(* Logix 5000 project; controller CarbonScout_MK6 vendor 1 type 14 code 154 rev 32.11; software revision 32.00; part 16 of 17 *)
(* tags used below, declared in another part *)
   ONS : BOOL[32];
   a_Software_Version : STRING;   // This must be updated and have a corrosponding change log and compadibility doc
   CS_DINTParams : DINT[100];
   CS_Seq : GEK_Sequence;
   CS_XRF : XRF;
   CS_XRF_Elements : LinearModelXRF;   // Linear model 0 is inital factory model and 1 is trimming model
   CS_XRF_Elements_Saved : LinearModelXRF;
   CS_XRF_RawModel : REAL[4];
   N50 : DINT[20];   // Out To Client (Ready only)
   NetworkHealthy : DINT;
   Oneshot3 : DINT;
   PLC_Powered : BOOL;
   Powered_Up : TIMER;
   Reg_Model : REAL[4];   // Calculated model output and site model
   Simulation : DINT;
   TimeAndDate : DINT[7];
   TimeAndDateW : DINT[7];
   Uptime : DINT;   // sec
   Valve_XV_01 : P_ValveSO;   // Sample Valve Tank 1
   Valve_XV_02 : P_ValveSO;   // Sample Valve Tank 2
   Valve_XV_03 : P_ValveSO;   // Sample Valve Tank 3
   Valve_XV_04 : P_ValveSO;   // Sample Valve Tank 4
   Valve_XV_05 : P_ValveSO;   // Sample Valve Tank 5
   Valve_XV_06 : P_ValveSO;   // Sample Valve Tank 6
   Valve_XV_07 : P_ValveSO;   // Sample Valve Tank 7
   Valve_XV_08 : P_ValveSO;   // Sample Valve Tank 8
   Valve_XV_09 : P_ValveSO;   // Sample Valve Tank 9
   Valve_XV_10 : P_ValveSO;   // Sample Valve Tank 10
   Valve_XV_11 : P_ValveSO;   // Purge Valve
   Valve_XV_12 : P_ValveSO;   // Slurry inlet vavle
   Valve_XV_13 : P_ValveSO;   // Sample line vavle
   XRF_RAWDINT : DINT[100];
(* SeqProgram, continued *)

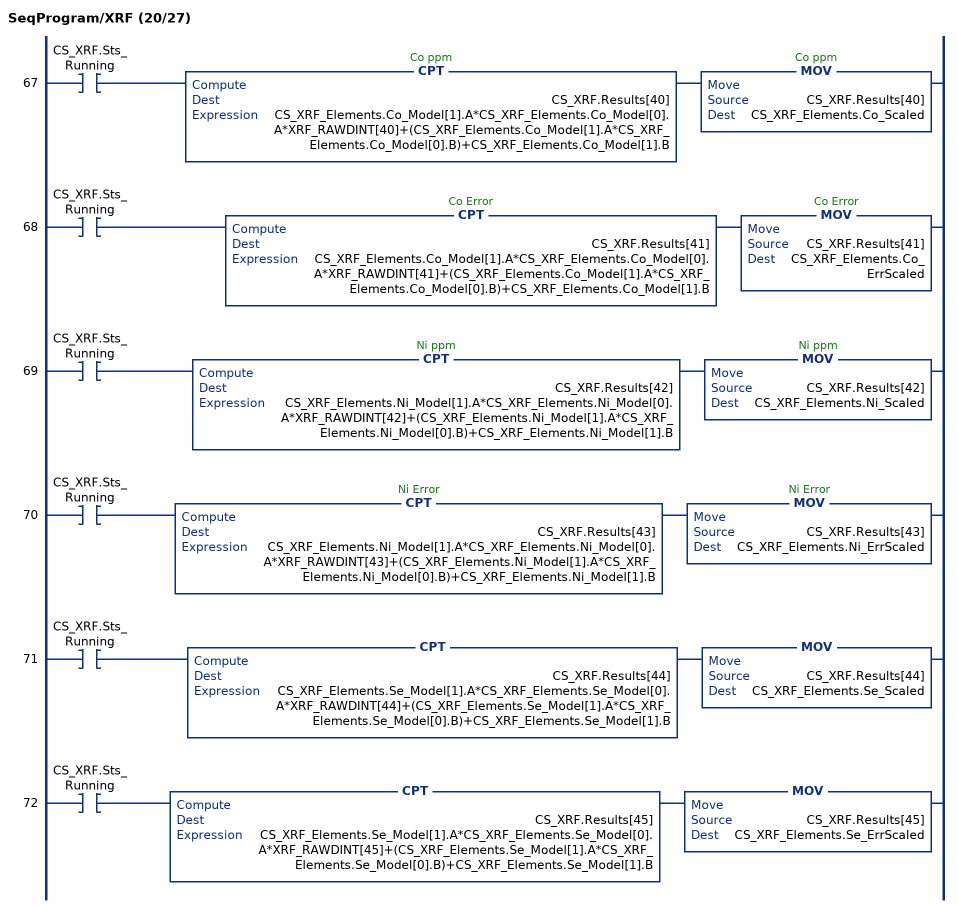
   67: XIC(CS_XRF.Sts_Running)CPT(CS_XRF.Results[40],CS_XRF_Elements.Co_Model[1].A*CS_XRF_Elements.Co_Model[0].A*XRF_RAWDINT[40]+(CS_XRF_Elements.Co_Model[1].A*CS_XRF_Elements.Co_Model[0].B)+CS_XRF_Elements.Co_Model[1].B)MOV(CS_XRF.Results[40],CS_XRF_Elements.Co_Scaled);
   68: XIC(CS_XRF.Sts_Running)CPT(CS_XRF.Results[41],CS_XRF_Elements.Co_Model[1].A*CS_XRF_Elements.Co_Model[0].A*XRF_RAWDINT[41]+(CS_XRF_Elements.Co_Model[1].A*CS_XRF_Elements.Co_Model[0].B)+CS_XRF_Elements.Co_Model[1].B)MOV(CS_XRF.Results[41],CS_XRF_Elements.Co_ErrScaled);
   69: XIC(CS_XRF.Sts_Running)CPT(CS_XRF.Results[42],CS_XRF_Elements.Ni_Model[1].A*CS_XRF_Elements.Ni_Model[0].A*XRF_RAWDINT[42]+(CS_XRF_Elements.Ni_Model[1].A*CS_XRF_Elements.Ni_Model[0].B)+CS_XRF_Elements.Ni_Model[1].B)MOV(CS_XRF.Results[42],CS_XRF_Elements.Ni_Scaled);
   70: XIC(CS_XRF.Sts_Running)CPT(CS_XRF.Results[43],CS_XRF_Elements.Ni_Model[1].A*CS_XRF_Elements.Ni_Model[0].A*XRF_RAWDINT[43]+(CS_XRF_Elements.Ni_Model[1].A*CS_XRF_Elements.Ni_Model[0].B)+CS_XRF_Elements.Ni_Model[1].B)MOV(CS_XRF.Results[43],CS_XRF_Elements.Ni_ErrScaled);
   71: XIC(CS_XRF.Sts_Running)CPT(CS_XRF.Results[44],CS_XRF_Elements.Se_Model[1].A*CS_XRF_Elements.Se_Model[0].A*XRF_RAWDINT[44]+(CS_XRF_Elements.Se_Model[1].A*CS_XRF_Elements.Se_Model[0].B)+CS_XRF_Elements.Se_Model[1].B)MOV(CS_XRF.Results[44],CS_XRF_Elements.Se_Scaled);
   72: XIC(CS_XRF.Sts_Running)CPT(CS_XRF.Results[45],CS_XRF_Elements.Se_Model[1].A*CS_XRF_Elements.Se_Model[0].A*XRF_RAWDINT[45]+(CS_XRF_Elements.Se_Model[1].A*CS_XRF_Elements.Se_Model[0].B)+CS_XRF_Elements.Se_Model[1].B)MOV(CS_XRF.Results[45],CS_XRF_Elements.Se_ErrScaled);
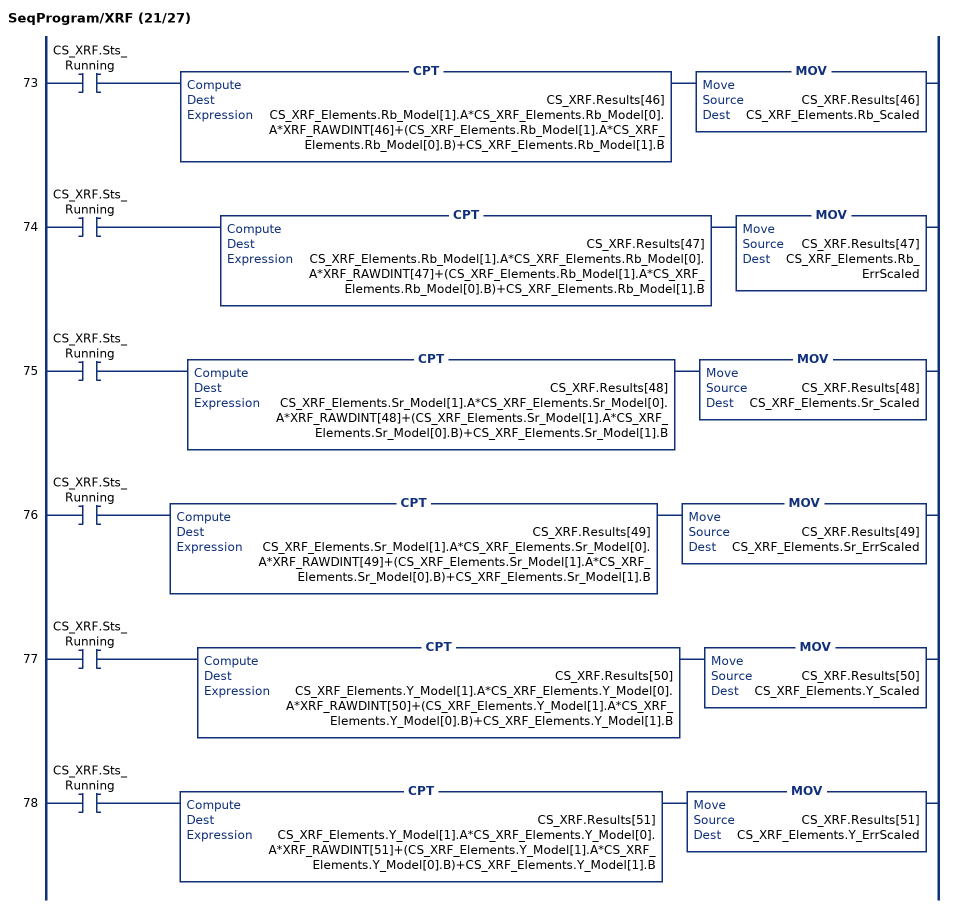
   73: XIC(CS_XRF.Sts_Running)CPT(CS_XRF.Results[46],CS_XRF_Elements.Rb_Model[1].A*CS_XRF_Elements.Rb_Model[0].A*XRF_RAWDINT[46]+(CS_XRF_Elements.Rb_Model[1].A*CS_XRF_Elements.Rb_Model[0].B)+CS_XRF_Elements.Rb_Model[1].B)MOV(CS_XRF.Results[46],CS_XRF_Elements.Rb_Scaled);
   74: XIC(CS_XRF.Sts_Running)CPT(CS_XRF.Results[47],CS_XRF_Elements.Rb_Model[1].A*CS_XRF_Elements.Rb_Model[0].A*XRF_RAWDINT[47]+(CS_XRF_Elements.Rb_Model[1].A*CS_XRF_Elements.Rb_Model[0].B)+CS_XRF_Elements.Rb_Model[1].B)MOV(CS_XRF.Results[47],CS_XRF_Elements.Rb_ErrScaled);
   75: XIC(CS_XRF.Sts_Running)CPT(CS_XRF.Results[48],CS_XRF_Elements.Sr_Model[1].A*CS_XRF_Elements.Sr_Model[0].A*XRF_RAWDINT[48]+(CS_XRF_Elements.Sr_Model[1].A*CS_XRF_Elements.Sr_Model[0].B)+CS_XRF_Elements.Sr_Model[1].B)MOV(CS_XRF.Results[48],CS_XRF_Elements.Sr_Scaled);
   76: XIC(CS_XRF.Sts_Running)CPT(CS_XRF.Results[49],CS_XRF_Elements.Sr_Model[1].A*CS_XRF_Elements.Sr_Model[0].A*XRF_RAWDINT[49]+(CS_XRF_Elements.Sr_Model[1].A*CS_XRF_Elements.Sr_Model[0].B)+CS_XRF_Elements.Sr_Model[1].B)MOV(CS_XRF.Results[49],CS_XRF_Elements.Sr_ErrScaled);
   77: XIC(CS_XRF.Sts_Running)CPT(CS_XRF.Results[50],CS_XRF_Elements.Y_Model[1].A*CS_XRF_Elements.Y_Model[0].A*XRF_RAWDINT[50]+(CS_XRF_Elements.Y_Model[1].A*CS_XRF_Elements.Y_Model[0].B)+CS_XRF_Elements.Y_Model[1].B)MOV(CS_XRF.Results[50],CS_XRF_Elements.Y_Scaled);
   78: XIC(CS_XRF.Sts_Running)CPT(CS_XRF.Results[51],CS_XRF_Elements.Y_Model[1].A*CS_XRF_Elements.Y_Model[0].A*XRF_RAWDINT[51]+(CS_XRF_Elements.Y_Model[1].A*CS_XRF_Elements.Y_Model[0].B)+CS_XRF_Elements.Y_Model[1].B)MOV(CS_XRF.Results[51],CS_XRF_Elements.Y_ErrScaled);
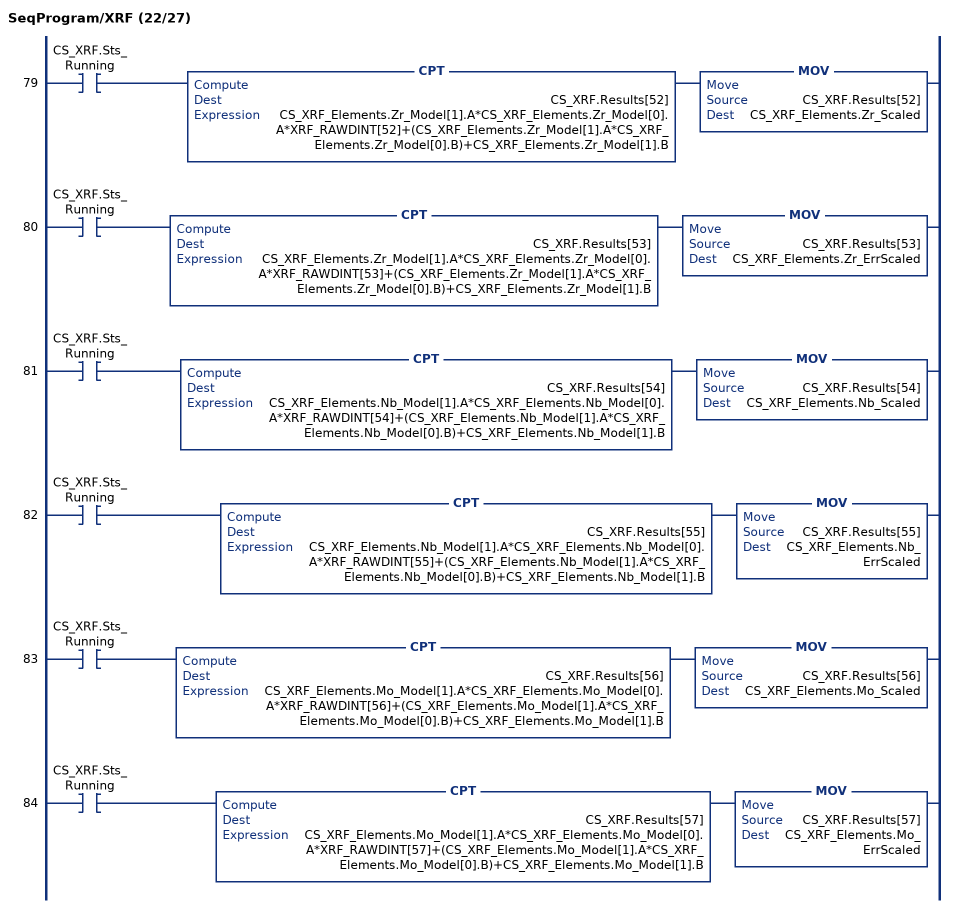
   79: XIC(CS_XRF.Sts_Running)CPT(CS_XRF.Results[52],CS_XRF_Elements.Zr_Model[1].A*CS_XRF_Elements.Zr_Model[0].A*XRF_RAWDINT[52]+(CS_XRF_Elements.Zr_Model[1].A*CS_XRF_Elements.Zr_Model[0].B)+CS_XRF_Elements.Zr_Model[1].B)MOV(CS_XRF.Results[52],CS_XRF_Elements.Zr_Scaled);
   80: XIC(CS_XRF.Sts_Running)CPT(CS_XRF.Results[53],CS_XRF_Elements.Zr_Model[1].A*CS_XRF_Elements.Zr_Model[0].A*XRF_RAWDINT[53]+(CS_XRF_Elements.Zr_Model[1].A*CS_XRF_Elements.Zr_Model[0].B)+CS_XRF_Elements.Zr_Model[1].B)MOV(CS_XRF.Results[53],CS_XRF_Elements.Zr_ErrScaled);
   81: XIC(CS_XRF.Sts_Running)CPT(CS_XRF.Results[54],CS_XRF_Elements.Nb_Model[1].A*CS_XRF_Elements.Nb_Model[0].A*XRF_RAWDINT[54]+(CS_XRF_Elements.Nb_Model[1].A*CS_XRF_Elements.Nb_Model[0].B)+CS_XRF_Elements.Nb_Model[1].B)MOV(CS_XRF.Results[54],CS_XRF_Elements.Nb_Scaled);
   82: XIC(CS_XRF.Sts_Running)CPT(CS_XRF.Results[55],CS_XRF_Elements.Nb_Model[1].A*CS_XRF_Elements.Nb_Model[0].A*XRF_RAWDINT[55]+(CS_XRF_Elements.Nb_Model[1].A*CS_XRF_Elements.Nb_Model[0].B)+CS_XRF_Elements.Nb_Model[1].B)MOV(CS_XRF.Results[55],CS_XRF_Elements.Nb_ErrScaled);
   83: XIC(CS_XRF.Sts_Running)CPT(CS_XRF.Results[56],CS_XRF_Elements.Mo_Model[1].A*CS_XRF_Elements.Mo_Model[0].A*XRF_RAWDINT[56]+(CS_XRF_Elements.Mo_Model[1].A*CS_XRF_Elements.Mo_Model[0].B)+CS_XRF_Elements.Mo_Model[1].B)MOV(CS_XRF.Results[56],CS_XRF_Elements.Mo_Scaled);
   84: XIC(CS_XRF.Sts_Running)CPT(CS_XRF.Results[57],CS_XRF_Elements.Mo_Model[1].A*CS_XRF_Elements.Mo_Model[0].A*XRF_RAWDINT[57]+(CS_XRF_Elements.Mo_Model[1].A*CS_XRF_Elements.Mo_Model[0].B)+CS_XRF_Elements.Mo_Model[1].B)MOV(CS_XRF.Results[57],CS_XRF_Elements.Mo_ErrScaled);
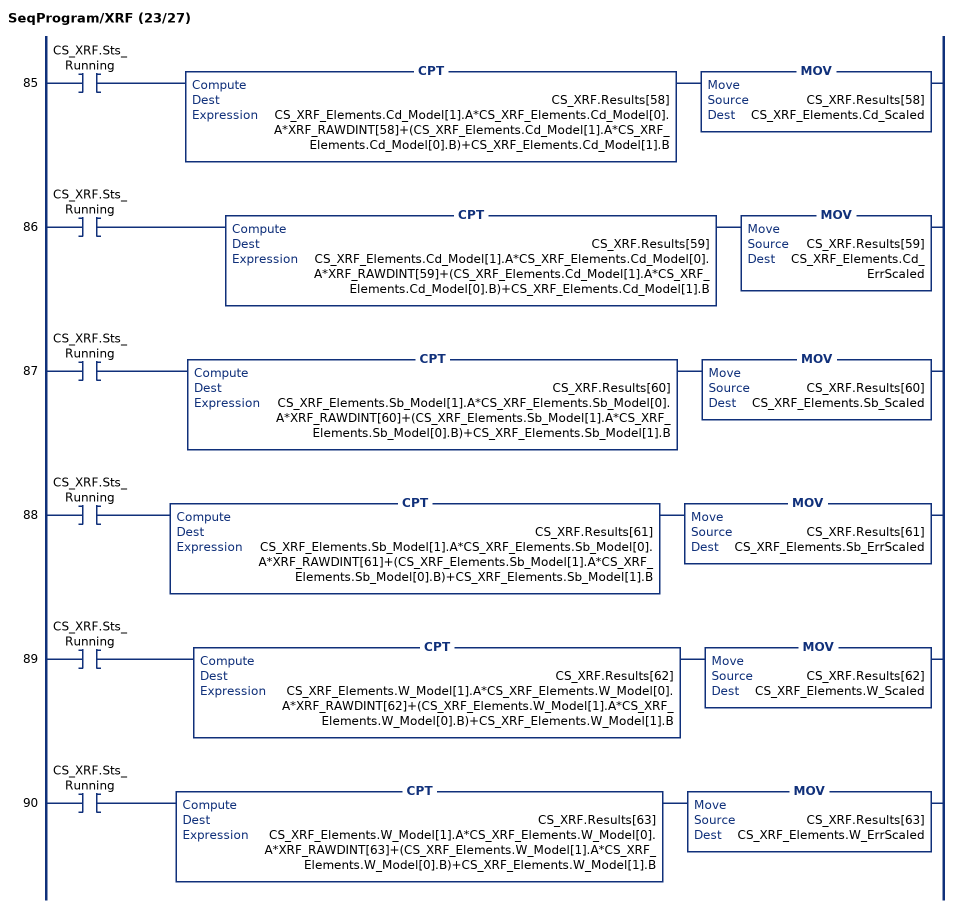
   85: XIC(CS_XRF.Sts_Running)CPT(CS_XRF.Results[58],CS_XRF_Elements.Cd_Model[1].A*CS_XRF_Elements.Cd_Model[0].A*XRF_RAWDINT[58]+(CS_XRF_Elements.Cd_Model[1].A*CS_XRF_Elements.Cd_Model[0].B)+CS_XRF_Elements.Cd_Model[1].B)MOV(CS_XRF.Results[58],CS_XRF_Elements.Cd_Scaled);
   86: XIC(CS_XRF.Sts_Running)CPT(CS_XRF.Results[59],CS_XRF_Elements.Cd_Model[1].A*CS_XRF_Elements.Cd_Model[0].A*XRF_RAWDINT[59]+(CS_XRF_Elements.Cd_Model[1].A*CS_XRF_Elements.Cd_Model[0].B)+CS_XRF_Elements.Cd_Model[1].B)MOV(CS_XRF.Results[59],CS_XRF_Elements.Cd_ErrScaled);
   87: XIC(CS_XRF.Sts_Running)CPT(CS_XRF.Results[60],CS_XRF_Elements.Sb_Model[1].A*CS_XRF_Elements.Sb_Model[0].A*XRF_RAWDINT[60]+(CS_XRF_Elements.Sb_Model[1].A*CS_XRF_Elements.Sb_Model[0].B)+CS_XRF_Elements.Sb_Model[1].B)MOV(CS_XRF.Results[60],CS_XRF_Elements.Sb_Scaled);
   88: XIC(CS_XRF.Sts_Running)CPT(CS_XRF.Results[61],CS_XRF_Elements.Sb_Model[1].A*CS_XRF_Elements.Sb_Model[0].A*XRF_RAWDINT[61]+(CS_XRF_Elements.Sb_Model[1].A*CS_XRF_Elements.Sb_Model[0].B)+CS_XRF_Elements.Sb_Model[1].B)MOV(CS_XRF.Results[61],CS_XRF_Elements.Sb_ErrScaled);
   89: XIC(CS_XRF.Sts_Running)CPT(CS_XRF.Results[62],CS_XRF_Elements.W_Model[1].A*CS_XRF_Elements.W_Model[0].A*XRF_RAWDINT[62]+(CS_XRF_Elements.W_Model[1].A*CS_XRF_Elements.W_Model[0].B)+CS_XRF_Elements.W_Model[1].B)MOV(CS_XRF.Results[62],CS_XRF_Elements.W_Scaled);
   90: XIC(CS_XRF.Sts_Running)CPT(CS_XRF.Results[63],CS_XRF_Elements.W_Model[1].A*CS_XRF_Elements.W_Model[0].A*XRF_RAWDINT[63]+(CS_XRF_Elements.W_Model[1].A*CS_XRF_Elements.W_Model[0].B)+CS_XRF_Elements.W_Model[1].B)MOV(CS_XRF.Results[63],CS_XRF_Elements.W_ErrScaled);
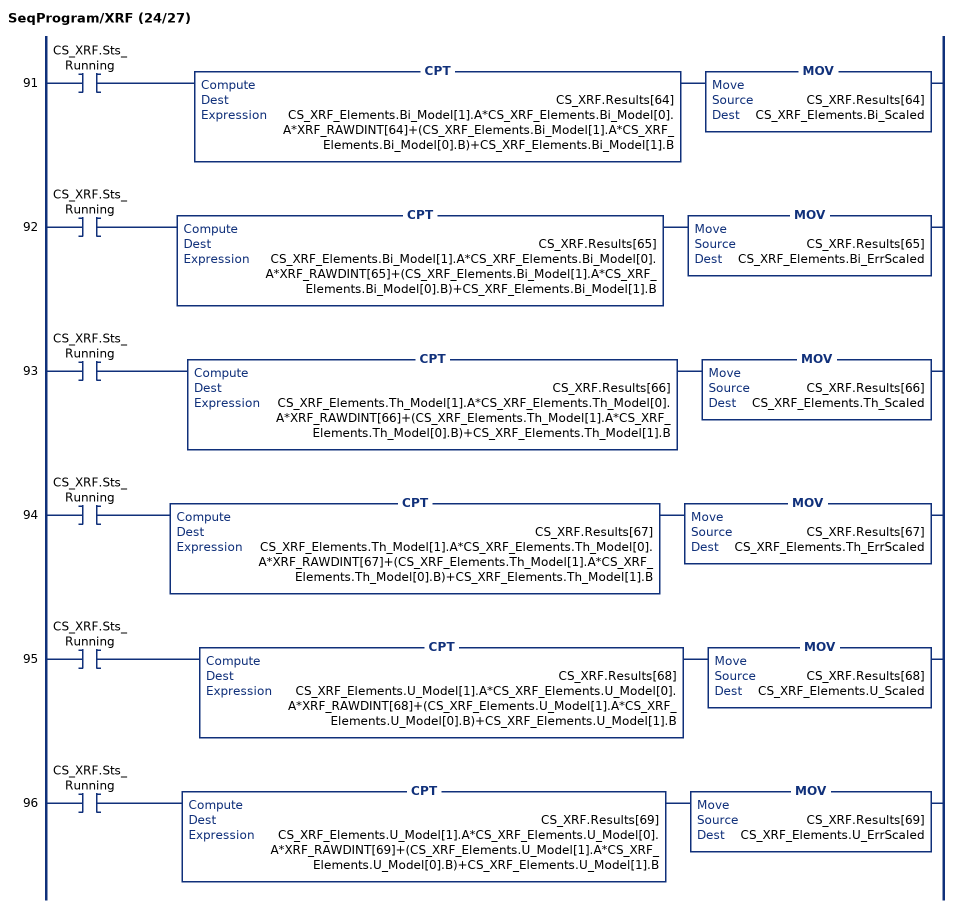
   91: XIC(CS_XRF.Sts_Running)CPT(CS_XRF.Results[64],CS_XRF_Elements.Bi_Model[1].A*CS_XRF_Elements.Bi_Model[0].A*XRF_RAWDINT[64]+(CS_XRF_Elements.Bi_Model[1].A*CS_XRF_Elements.Bi_Model[0].B)+CS_XRF_Elements.Bi_Model[1].B)MOV(CS_XRF.Results[64],CS_XRF_Elements.Bi_Scaled);
   92: XIC(CS_XRF.Sts_Running)CPT(CS_XRF.Results[65],CS_XRF_Elements.Bi_Model[1].A*CS_XRF_Elements.Bi_Model[0].A*XRF_RAWDINT[65]+(CS_XRF_Elements.Bi_Model[1].A*CS_XRF_Elements.Bi_Model[0].B)+CS_XRF_Elements.Bi_Model[1].B)MOV(CS_XRF.Results[65],CS_XRF_Elements.Bi_ErrScaled);
   93: XIC(CS_XRF.Sts_Running)CPT(CS_XRF.Results[66],CS_XRF_Elements.Th_Model[1].A*CS_XRF_Elements.Th_Model[0].A*XRF_RAWDINT[66]+(CS_XRF_Elements.Th_Model[1].A*CS_XRF_Elements.Th_Model[0].B)+CS_XRF_Elements.Th_Model[1].B)MOV(CS_XRF.Results[66],CS_XRF_Elements.Th_Scaled);
   94: XIC(CS_XRF.Sts_Running)CPT(CS_XRF.Results[67],CS_XRF_Elements.Th_Model[1].A*CS_XRF_Elements.Th_Model[0].A*XRF_RAWDINT[67]+(CS_XRF_Elements.Th_Model[1].A*CS_XRF_Elements.Th_Model[0].B)+CS_XRF_Elements.Th_Model[1].B)MOV(CS_XRF.Results[67],CS_XRF_Elements.Th_ErrScaled);
   95: XIC(CS_XRF.Sts_Running)CPT(CS_XRF.Results[68],CS_XRF_Elements.U_Model[1].A*CS_XRF_Elements.U_Model[0].A*XRF_RAWDINT[68]+(CS_XRF_Elements.U_Model[1].A*CS_XRF_Elements.U_Model[0].B)+CS_XRF_Elements.U_Model[1].B)MOV(CS_XRF.Results[68],CS_XRF_Elements.U_Scaled);
   96: XIC(CS_XRF.Sts_Running)CPT(CS_XRF.Results[69],CS_XRF_Elements.U_Model[1].A*CS_XRF_Elements.U_Model[0].A*XRF_RAWDINT[69]+(CS_XRF_Elements.U_Model[1].A*CS_XRF_Elements.U_Model[0].B)+CS_XRF_Elements.U_Model[1].B)MOV(CS_XRF.Results[69],CS_XRF_Elements.U_ErrScaled);
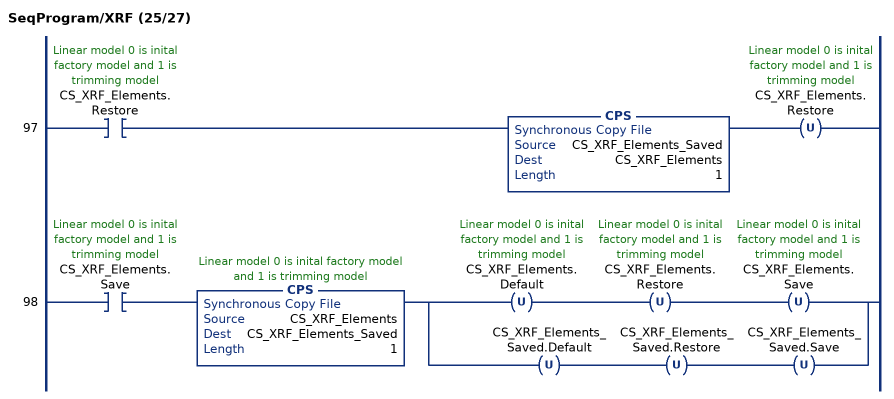
   97: XIC(CS_XRF_Elements.Restore)CPS(CS_XRF_Elements_Saved,CS_XRF_Elements,1)OTU(CS_XRF_Elements.Restore);
   98: XIC(CS_XRF_Elements.Save)CPS(CS_XRF_Elements,CS_XRF_Elements_Saved,1)[OTU(CS_XRF_Elements.Default) OTU(CS_XRF_Elements.Restore) OTU(CS_XRF_Elements.Save) ,OTU(CS_XRF_Elements_Saved.Default) OTU(CS_XRF_Elements_Saved.Restore) OTU(CS_XRF_Elements_Saved.Save) ];
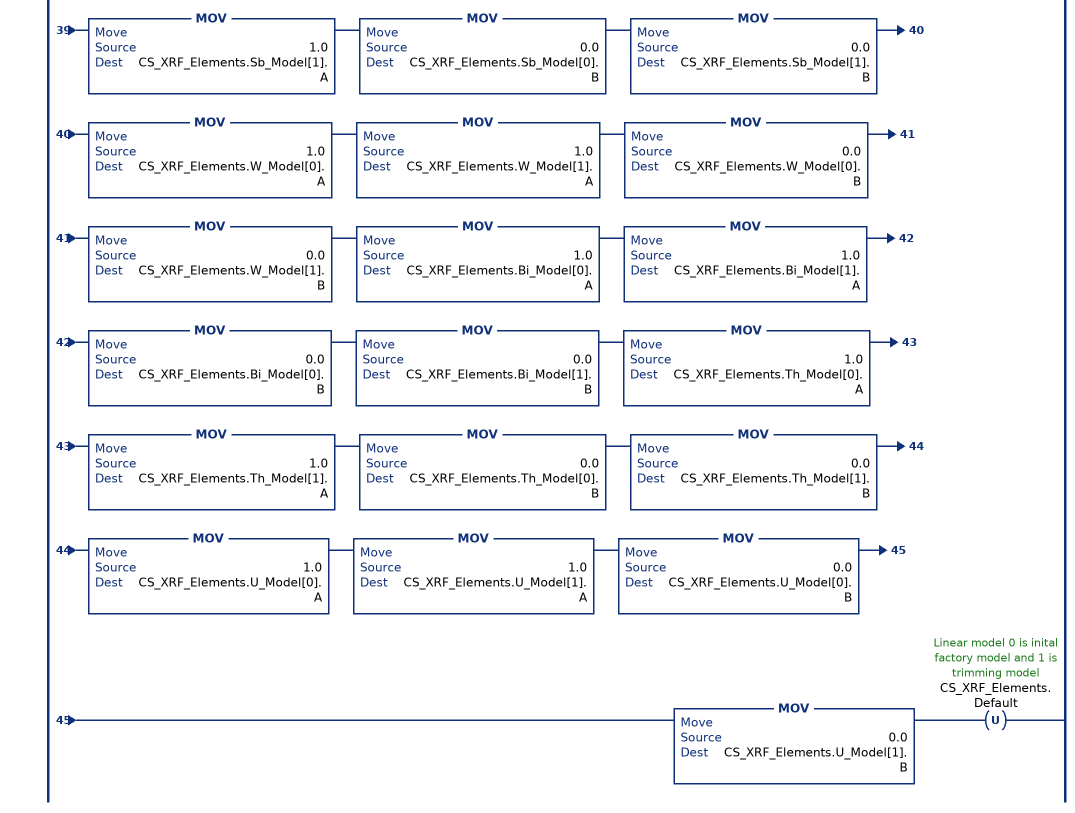
   // Default Settings
   // No cal model
   99: XIC(CS_XRF_Elements.Default)MOV(1.0,CS_XRF_Elements.Au_Model[0].A)MOV(1.0,CS_XRF_Elements.Au_Model[1].A)MOV(0.0,CS_XRF_Elements.Au_Model[0].B)MOV(0.0,CS_XRF_Elements.Au_Model[1].B)MOV(1.0,CS_XRF_Elements.As_Model[0].A)MOV(1.0,CS_XRF_Elements.As_Model[1].A)MOV(0.0,CS_XRF_Elements.As_Model[0].B)MOV(0.0,CS_XRF_Elements.As_Model[1].B)MOV(1.0,CS_XRF_Elements.Cu_Model[0].A)MOV(1.0,CS_XRF_Elements.Cu_Model[1].A)MOV(0.0,CS_XRF_Elements.Cu_Model[0].B)MOV(0.0,CS_XRF_Elements.Cu_Model[1].B)MOV(1.0,CS_XRF_Elements.Fe_Model[0].A)MOV(1.0,CS_XRF_Elements.Fe_Model[1].A)MOV(0.0,CS_XRF_Elements.Fe_Model[0].B)MOV(0.0,CS_XRF_Elements.Fe_Model[1].B)MOV(1.0,CS_XRF_Elements.Ag_Model[0].A)MOV(1.0,CS_XRF_Elements.Ag_Model[1].A)MOV(0.0,CS_XRF_Elements.Ag_Model[0].B)MOV(0.0,CS_XRF_Elements.Ag_Model[1].B)MOV(1.0,CS_XRF_Elements.Hg_Model[0].A)MOV(1.0,CS_XRF_Elements.Hg_Model[1].A)MOV(0.0,CS_XRF_Elements.Hg_Model[0].B)MOV(0.0,CS_XRF_Elements.Hg_Model[1].B)MOV(1.0,CS_XRF_Elements.Pb_Model[0].A)MOV(1.0,CS_XRF_Elements.Pb_Model[1].A)MOV(0.0,CS_XRF_Elements.Pb_Model[0].B)MOV(0.0,CS_XRF_Elements.Pb_Model[1].B)MOV(1.0,CS_XRF_Elements.Zn_Model[0].A)MOV(1.0,CS_XRF_Elements.Zn_Model[1].A)MOV(0.0,CS_XRF_Elements.Zn_Model[0].B)MOV(0.0,CS_XRF_Elements.Zn_Model[1].B)MOV(1.0,CS_XRF_Elements.Sn_Model[0].A)MOV(1.0,CS_XRF_Elements.Sn_Model[1].A)MOV(0.0,CS_XRF_Elements.Sn_Model[0].B)MOV(0.0,CS_XRF_Elements.Sn_Model[1].B)MOV(1.0,CS_XRF_Elements.Ca_Model[0].A)MOV(1.0,CS_XRF_Elements.Ca_Model[1].A)MOV(0.0,CS_XRF_Elements.Ca_Model[0].B)MOV(0.0,CS_XRF_Elements.Ca_Model[1].B)MOV(1.0,CS_XRF_Elements.Mg_Model[0].A)MOV(1.0,CS_XRF_Elements.Mg_Model[1].A)MOV(0.0,CS_XRF_Elements.Mg_Model[0].B)MOV(0.0,CS_XRF_Elements.Mg_Model[1].B)MOV(1.0,CS_XRF_Elements.Al_Model[0].A)MOV(1.0,CS_XRF_Elements.Al_Model[1].A)MOV(0.0,CS_XRF_Elements.Al_Model[0].B)MOV(0.0,CS_XRF_Elements.Al_Model[1].B)MOV(1.0,CS_XRF_Elements.Si_Model[0].A)MOV(1.0,CS_XRF_Elements.Si_Model[1].A)MOV(0.0,CS_XRF_Elements.Si_Model[0].B)MOV(0.0,CS_XRF_Elements.Si_Model[1].B)MOV(1.0,CS_XRF_Elements.S_Model[0].A)MOV(1.0,CS_XRF_Elements.S_Model[1].A)MOV(0.0,CS_XRF_Elements.S_Model[0].B)MOV(0.0,CS_XRF_Elements.S_Model[1].B)MOV(1.0,CS_XRF_Elements.K_Model[0].A)MOV(1.0,CS_XRF_Elements.K_Model[1].A)MOV(0.0,CS_XRF_Elements.K_Model[0].B)MOV(0.0,CS_XRF_Elements.K_Model[1].B)MOV(1.0,CS_XRF_Elements.Ti_Model[0].A)MOV(1.0,CS_XRF_Elements.Ti_Model[1].A)MOV(0.0,CS_XRF_Elements.Ti_Model[0].B)MOV(0.0,CS_XRF_Elements.Ti_Model[1].B)MOV(1.0,CS_XRF_Elements.V_Model[0].A)MOV(1.0,CS_XRF_Elements.V_Model[1].A)MOV(0.0,CS_XRF_Elements.V_Model[0].B)MOV(0.0,CS_XRF_Elements.V_Model[1].B)MOV(1.0,CS_XRF_Elements.Cr_Model[0].A)MOV(1.0,CS_XRF_Elements.Cr_Model[1].A)MOV(0.0,CS_XRF_Elements.Cr_Model[0].B)MOV(0.0,CS_XRF_Elements.Cr_Model[1].B)MOV(1.0,CS_XRF_Elements.Mn_Model[0].A)MOV(1.0,CS_XRF_Elements.Mn_Model[1].A)MOV(0.0,CS_XRF_Elements.Mn_Model[0].B)MOV(0.0,CS_XRF_Elements.Mn_Model[1].B)MOV(1.0,CS_XRF_Elements.Co_Model[0].A)MOV(1.0,CS_XRF_Elements.Co_Model[1].A)MOV(0.0,CS_XRF_Elements.Co_Model[0].B)MOV(0.0,CS_XRF_Elements.Co_Model[1].B)MOV(1.0,CS_XRF_Elements.Ni_Model[0].A)MOV(1.0,CS_XRF_Elements.Ni_Model[1].A)MOV(0.0,CS_XRF_Elements.Ni_Model[0].B)MOV(0.0,CS_XRF_Elements.Ni_Model[1].B)MOV(1.0,CS_XRF_Elements.Se_Model[0].A)MOV(1.0,CS_XRF_Elements.Se_Model[1].A)MOV(0.0,CS_XRF_Elements.Se_Model[0].B)MOV(0.0,CS_XRF_Elements.Se_Model[1].B)MOV(1.0,CS_XRF_Elements.Rb_Model[0].A)MOV(1.0,CS_XRF_Elements.Rb_Model[1].A)MOV(0.0,CS_XRF_Elements.Rb_Model[0].B)MOV(0.0,CS_XRF_Elements.Rb_Model[1].B)MOV(1.0,CS_XRF_Elements.Sr_Model[0].A)MOV(1.0,CS_XRF_Elements.Sr_Model[1].A)MOV(0.0,CS_XRF_Elements.Sr_Model[0].B)MOV(0.0,CS_XRF_Elements.Sr_Model[1].B)MOV(1.0,CS_XRF_Elements.Y_Model[0].A)MOV(1.0,CS_XRF_Elements.Y_Model[1].A)MOV(0.0,CS_XRF_Elements.Y_Model[0].B)MOV(0.0,CS_XRF_Elements.Y_Model[1].B)MOV(1.0,CS_XRF_Elements.Zr_Model[0].A)MOV(1.0,CS_XRF_Elements.Zr_Model[1].A)MOV(0.0,CS_XRF_Elements.Zr_Model[0].B)MOV(0.0,CS_XRF_Elements.Zr_Model[1].B)MOV(1.0,CS_XRF_Elements.Nb_Model[0].A)MOV(1.0,CS_XRF_Elements.Nb_Model[1].A)MOV(0.0,CS_XRF_Elements.Nb_Model[0].B)MOV(0.0,CS_XRF_Elements.Nb_Model[1].B)MOV(1.0,CS_XRF_Elements.Mo_Model[0].A)MOV(1.0,CS_XRF_Elements.Mo_Model[1].A)MOV(0.0,CS_XRF_Elements.Mo_Model[0].B)MOV(0.0,CS_XRF_Elements.Mo_Model[1].B)MOV(1.0,CS_XRF_Elements.Cd_Model[0].A)MOV(1.0,CS_XRF_Elements.Cd_Model[1].A)MOV(0.0,CS_XRF_Elements.Cd_Model[0].B)MOV(0.0,CS_XRF_Elements.Cd_Model[1].B)MOV(1.0,CS_XRF_Elements.Sb_Model[0].A)MOV(1.0,CS_XRF_Elements.Sb_Model[1].A)MOV(0.0,CS_XRF_Elements.Sb_Model[0].B)MOV(0.0,CS_XRF_Elements.Sb_Model[1].B)MOV(1.0,CS_XRF_Elements.W_Model[0].A)MOV(1.0,CS_XRF_Elements.W_Model[1].A)MOV(0.0,CS_XRF_Elements.W_Model[0].B)MOV(0.0,CS_XRF_Elements.W_Model[1].B)MOV(1.0,CS_XRF_Elements.Bi_Model[0].A)MOV(1.0,CS_XRF_Elements.Bi_Model[1].A)MOV(0.0,CS_XRF_Elements.Bi_Model[0].B)MOV(0.0,CS_XRF_Elements.Bi_Model[1].B)MOV(1.0,CS_XRF_Elements.Th_Model[0].A)MOV(1.0,CS_XRF_Elements.Th_Model[1].A)MOV(0.0,CS_XRF_Elements.Th_Model[0].B)MOV(0.0,CS_XRF_Elements.Th_Model[1].B)MOV(1.0,CS_XRF_Elements.U_Model[0].A)MOV(1.0,CS_XRF_Elements.U_Model[1].A)MOV(0.0,CS_XRF_Elements.U_Model[0].B)MOV(0.0,CS_XRF_Elements.U_Model[1].B)OTU(CS_XRF_Elements.Default);
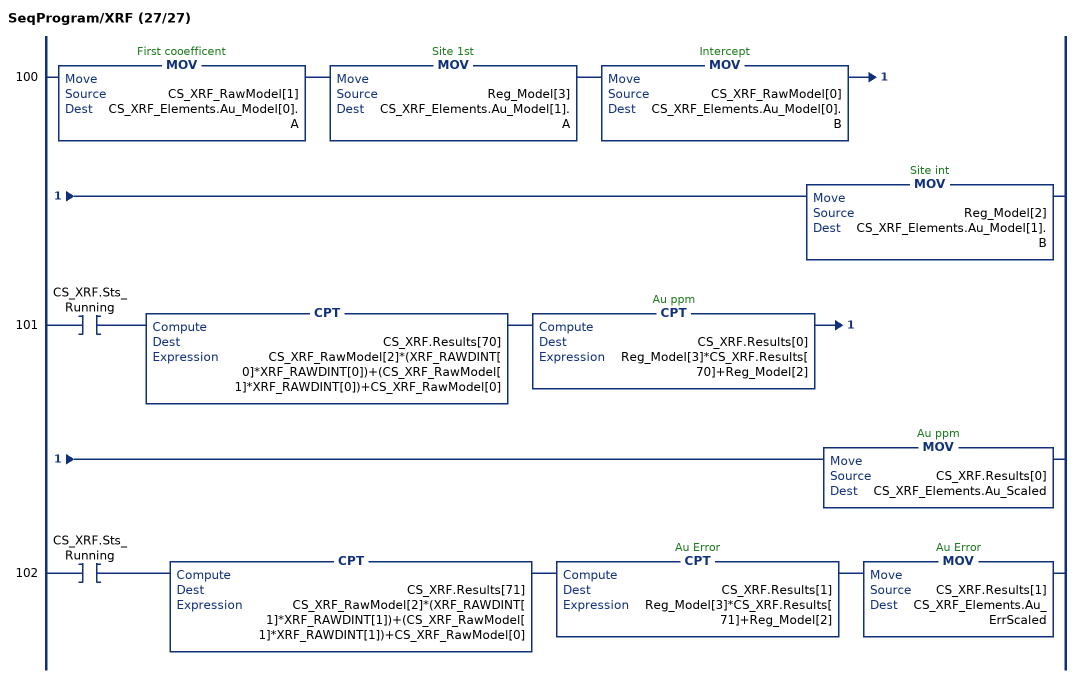
   100: MOV(CS_XRF_RawModel[1],CS_XRF_Elements.Au_Model[0].A)MOV(Reg_Model[3],CS_XRF_Elements.Au_Model[1].A)MOV(CS_XRF_RawModel[0],CS_XRF_Elements.Au_Model[0].B)MOV(Reg_Model[2],CS_XRF_Elements.Au_Model[1].B);
   101: XIC(CS_XRF.Sts_Running)CPT(CS_XRF.Results[70],CS_XRF_RawModel[2]*(XRF_RAWDINT[0]*XRF_RAWDINT[0])+(CS_XRF_RawModel[1]*XRF_RAWDINT[0])+CS_XRF_RawModel[0])CPT(CS_XRF.Results[0],Reg_Model[3]*CS_XRF.Results[70]+Reg_Model[2])MOV(CS_XRF.Results[0],CS_XRF_Elements.Au_Scaled);
   102: XIC(CS_XRF.Sts_Running)CPT(CS_XRF.Results[71],CS_XRF_RawModel[2]*(XRF_RAWDINT[1]*XRF_RAWDINT[1])+(CS_XRF_RawModel[1]*XRF_RAWDINT[1])+CS_XRF_RawModel[0])CPT(CS_XRF.Results[1],Reg_Model[3]*CS_XRF.Results[71]+Reg_Model[2])MOV(CS_XRF.Results[1],CS_XRF_Elements.Au_ErrScaled);
END_ROUTINE
END_PROGRAM

PROGRAM SystemTask   (* main routine Main *)
VAR
   zIO_EntryMasked : DINT := 4096;
   zIO_EntryStatus : DINT := 4096;
END_VAR

ROUTINE Main   (* ladder *)
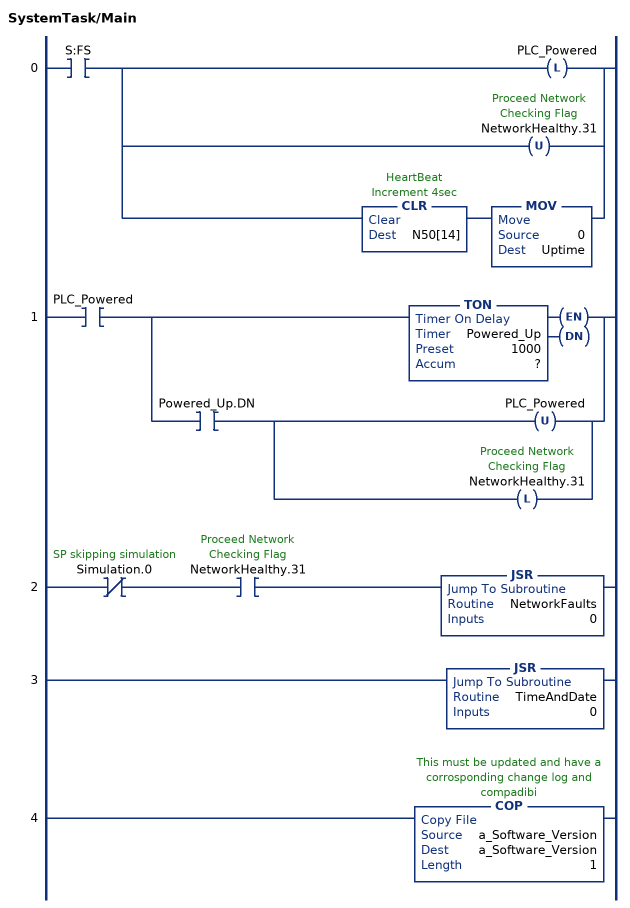
   0: XIC(S:FS)[OTL(PLC_Powered) ,OTU(NetworkHealthy.31) ,CLR(N50[14]) MOV(0,Uptime) ];
   1: XIC(PLC_Powered)[TON(Powered_Up,?,?) ,XIC(Powered_Up.DN) [OTU(PLC_Powered) ,OTL(NetworkHealthy.31) ] ];
   2: XIO(Simulation.0)XIC(NetworkHealthy.31)JSR(NetworkFaults,0);
   3: JSR(TimeAndDate,0);
   4: COP(a_Software_Version,a_Software_Version,1);
END_ROUTINE

ROUTINE NetworkFaults   (* ladder *)
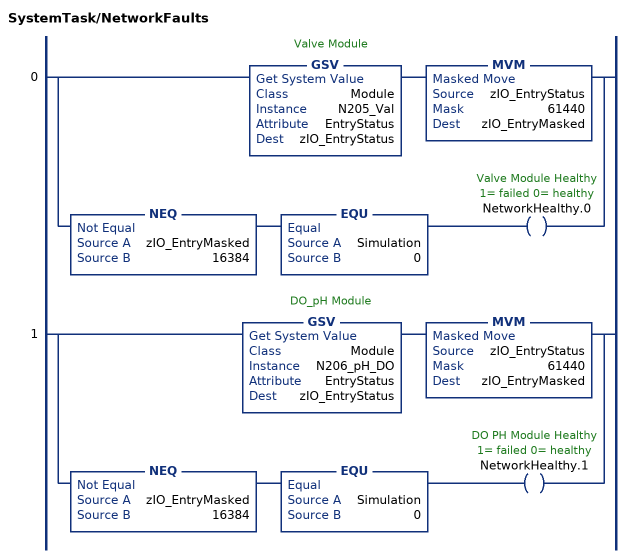
   // Valve Module
   0: [GSV(Module,N205_Val,EntryStatus,zIO_EntryStatus) MVM(zIO_EntryStatus,61440,zIO_EntryMasked) ,NEQ(zIO_EntryMasked,16384) EQU(Simulation,0) OTE(NetworkHealthy.0) ];
   // DO_pH Module
   1: [GSV(Module,N206_pH_DO,EntryStatus,zIO_EntryStatus) MVM(zIO_EntryStatus,61440,zIO_EntryMasked) ,NEQ(zIO_EntryMasked,16384) EQU(Simulation,0) OTE(NetworkHealthy.1) ];
END_ROUTINE

ROUTINE TimeAndDate   (* ladder *)
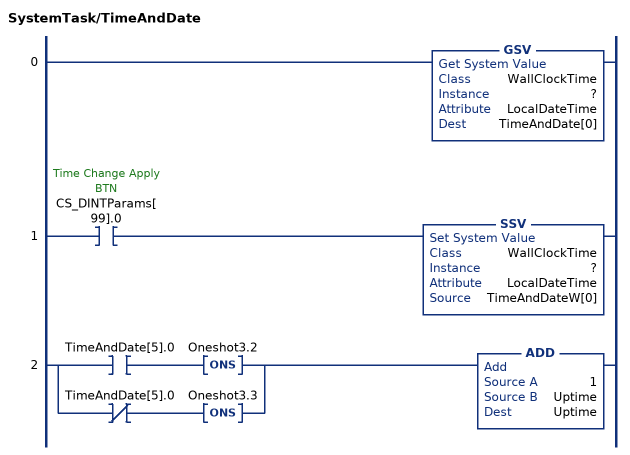
   0: GSV(WallClockTime,?,LocalDateTime,TimeAndDate[0]);
   1: XIC(CS_DINTParams[99].0)SSV(WallClockTime,?,LocalDateTime,TimeAndDateW[0]);
   2: [XIC(TimeAndDate[5].0) ONS(Oneshot3.2) ,XIO(TimeAndDate[5].0) ONS(Oneshot3.3) ]ADD(1,Uptime,Uptime);
END_ROUTINE
END_PROGRAM

PROGRAM Valves   (* main routine Main *)
VAR
   ValveOneshot : DINT;
END_VAR

ROUTINE Main   (* ladder *)
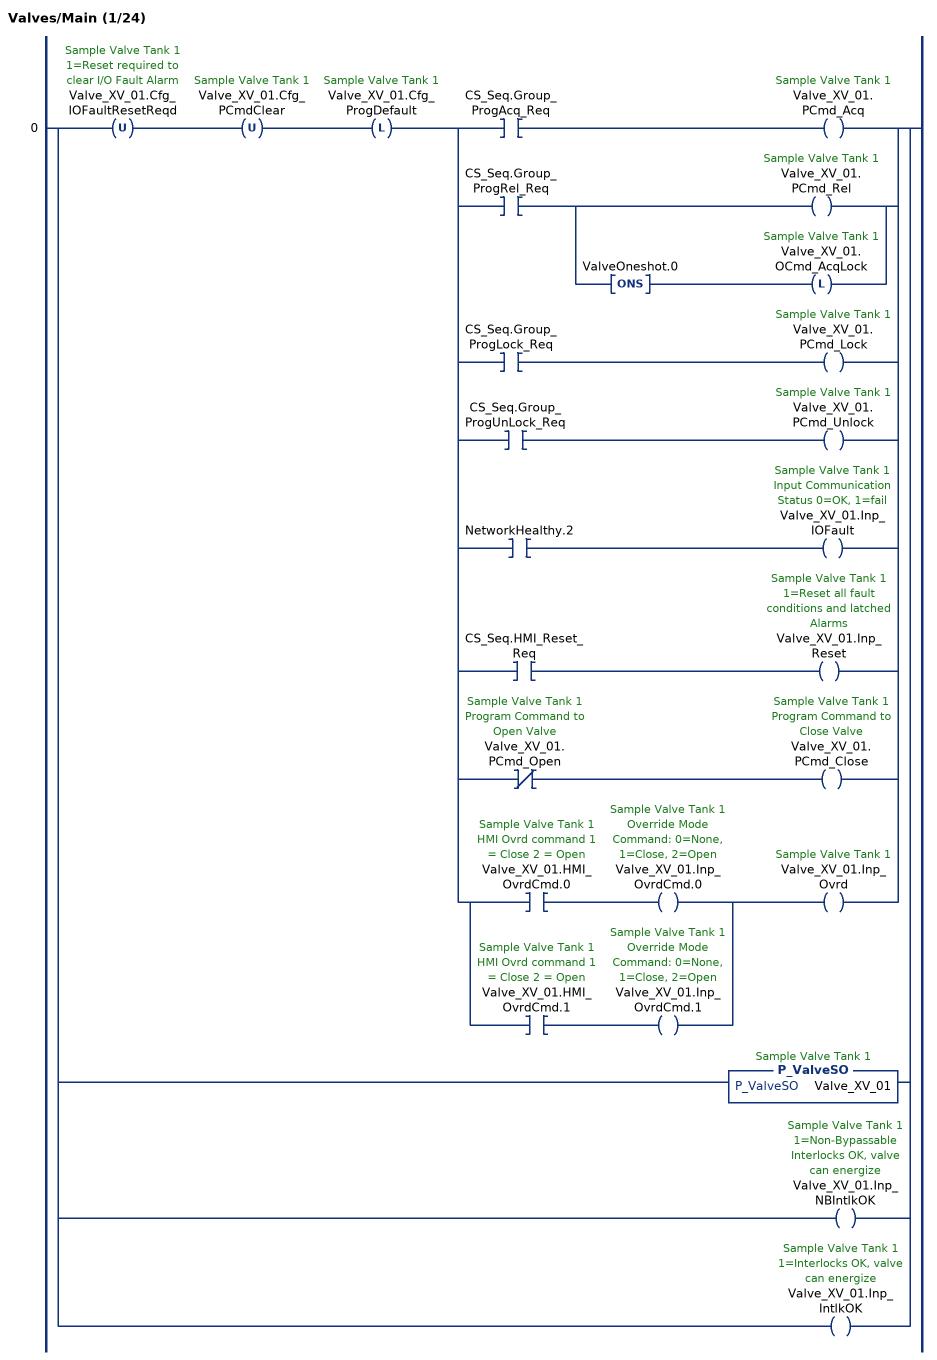
   0: [OTU(Valve_XV_01.Cfg_IOFaultResetReqd) OTU(Valve_XV_01.Cfg_PCmdClear) OTL(Valve_XV_01.Cfg_ProgDefault) [XIC(CS_Seq.Group_ProgAcq_Req) OTE(Valve_XV_01.PCmd_Acq) ,XIC(CS_Seq.Group_ProgRel_Req) [OTE(Valve_XV_01.PCmd_Rel) ,ONS(ValveOneshot.0) OTL(Valve_XV_01.OCmd_AcqLock) ] ,XIC(CS_Seq.Group_ProgLock_Req) OTE(Valve_XV_01.PCmd_Lock) ,XIC(CS_Seq.Group_ProgUnLock_Req) OTE(Valve_XV_01.PCmd_Unlock) ,XIC(NetworkHealthy.2) OTE(Valve_XV_01.Inp_IOFault) ,XIC(CS_Seq.HMI_Reset_Req) OTE(Valve_XV_01.Inp_Reset) ,XIO(Valve_XV_01.PCmd_Open) OTE(Valve_XV_01.PCmd_Close) ,[XIC(Valve_XV_01.HMI_OvrdCmd.0) OTE(Valve_XV_01.Inp_OvrdCmd.0) ,XIC(Valve_XV_01.HMI_OvrdCmd.1) OTE(Valve_XV_01.Inp_OvrdCmd.1) ] OTE(Valve_XV_01.Inp_Ovrd) ] ,[P_ValveSO(Valve_XV_01) ,OTE(Valve_XV_01.Inp_NBIntlkOK) ,OTE(Valve_XV_01.Inp_IntlkOK) ] ];
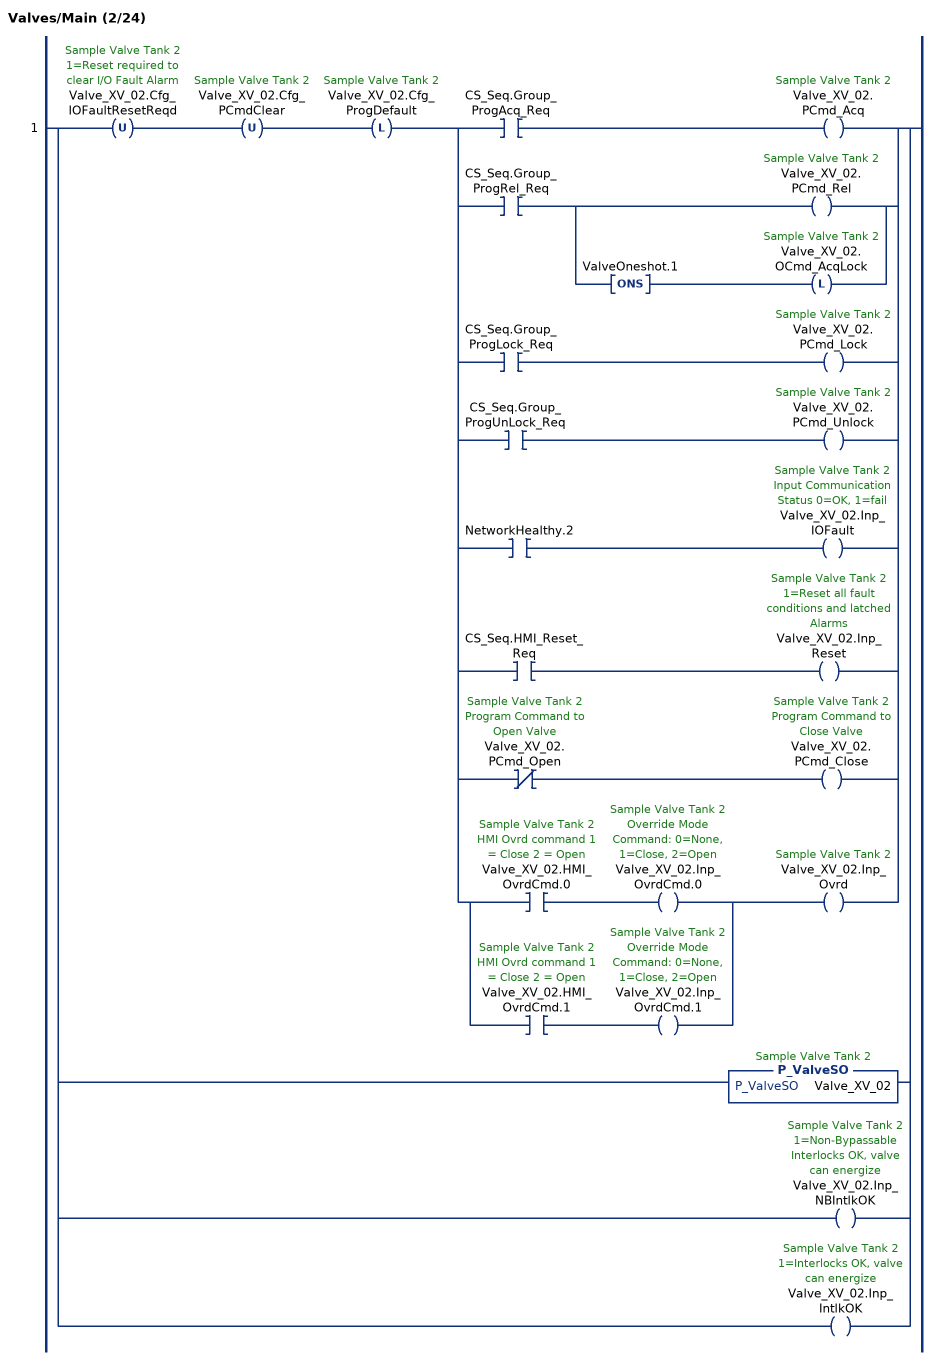
   1: [OTU(Valve_XV_02.Cfg_IOFaultResetReqd) OTU(Valve_XV_02.Cfg_PCmdClear) OTL(Valve_XV_02.Cfg_ProgDefault) [XIC(CS_Seq.Group_ProgAcq_Req) OTE(Valve_XV_02.PCmd_Acq) ,XIC(CS_Seq.Group_ProgRel_Req) [OTE(Valve_XV_02.PCmd_Rel) ,ONS(ValveOneshot.1) OTL(Valve_XV_02.OCmd_AcqLock) ] ,XIC(CS_Seq.Group_ProgLock_Req) OTE(Valve_XV_02.PCmd_Lock) ,XIC(CS_Seq.Group_ProgUnLock_Req) OTE(Valve_XV_02.PCmd_Unlock) ,XIC(NetworkHealthy.2) OTE(Valve_XV_02.Inp_IOFault) ,XIC(CS_Seq.HMI_Reset_Req) OTE(Valve_XV_02.Inp_Reset) ,XIO(Valve_XV_02.PCmd_Open) OTE(Valve_XV_02.PCmd_Close) ,[XIC(Valve_XV_02.HMI_OvrdCmd.0) OTE(Valve_XV_02.Inp_OvrdCmd.0) ,XIC(Valve_XV_02.HMI_OvrdCmd.1) OTE(Valve_XV_02.Inp_OvrdCmd.1) ] OTE(Valve_XV_02.Inp_Ovrd) ] ,[P_ValveSO(Valve_XV_02) ,OTE(Valve_XV_02.Inp_NBIntlkOK) ,OTE(Valve_XV_02.Inp_IntlkOK) ] ];
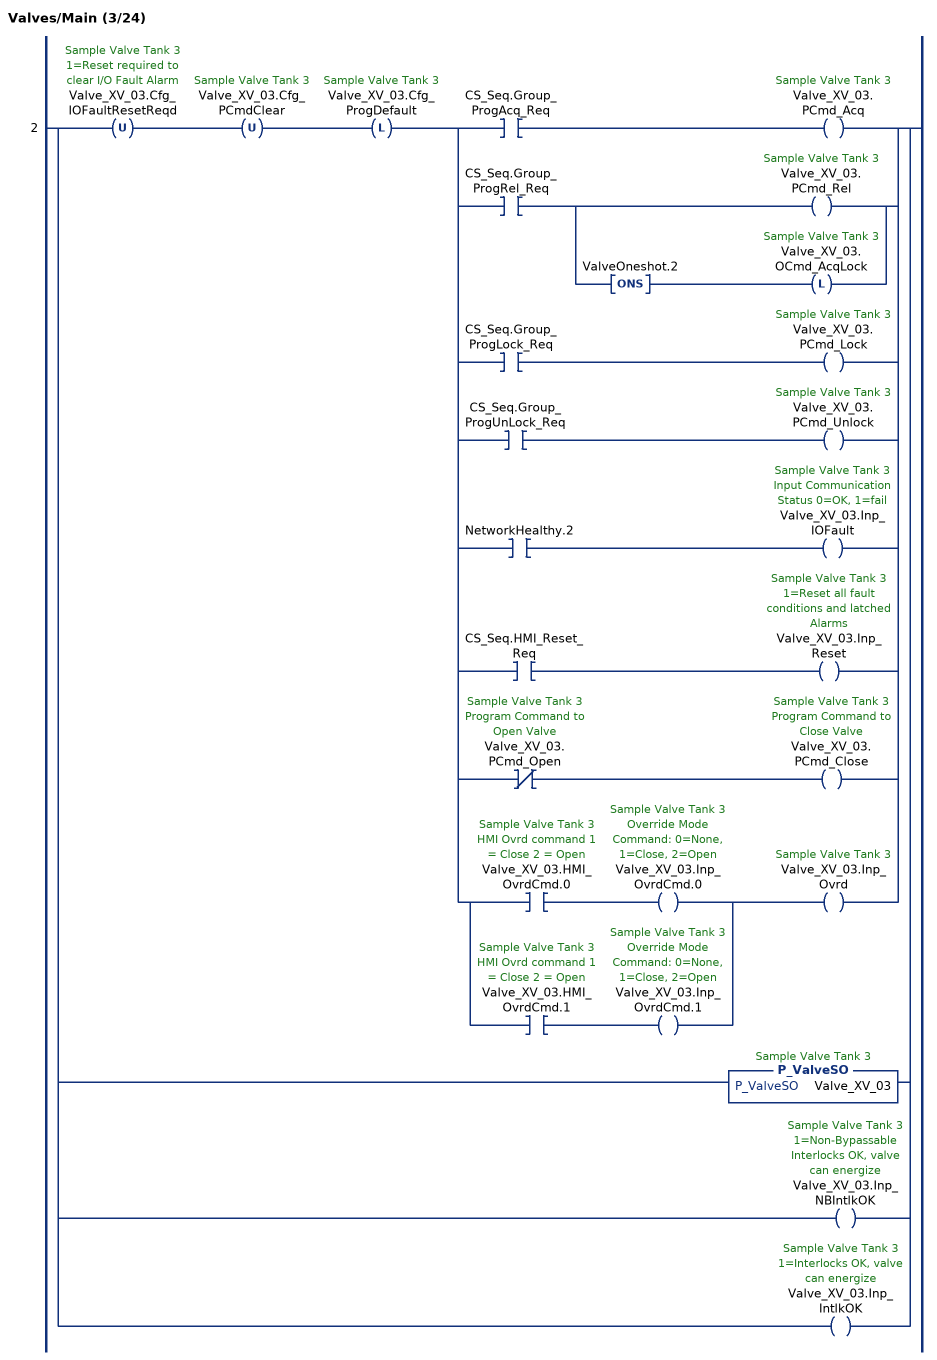
   2: [OTU(Valve_XV_03.Cfg_IOFaultResetReqd) OTU(Valve_XV_03.Cfg_PCmdClear) OTL(Valve_XV_03.Cfg_ProgDefault) [XIC(CS_Seq.Group_ProgAcq_Req) OTE(Valve_XV_03.PCmd_Acq) ,XIC(CS_Seq.Group_ProgRel_Req) [OTE(Valve_XV_03.PCmd_Rel) ,ONS(ValveOneshot.2) OTL(Valve_XV_03.OCmd_AcqLock) ] ,XIC(CS_Seq.Group_ProgLock_Req) OTE(Valve_XV_03.PCmd_Lock) ,XIC(CS_Seq.Group_ProgUnLock_Req) OTE(Valve_XV_03.PCmd_Unlock) ,XIC(NetworkHealthy.2) OTE(Valve_XV_03.Inp_IOFault) ,XIC(CS_Seq.HMI_Reset_Req) OTE(Valve_XV_03.Inp_Reset) ,XIO(Valve_XV_03.PCmd_Open) OTE(Valve_XV_03.PCmd_Close) ,[XIC(Valve_XV_03.HMI_OvrdCmd.0) OTE(Valve_XV_03.Inp_OvrdCmd.0) ,XIC(Valve_XV_03.HMI_OvrdCmd.1) OTE(Valve_XV_03.Inp_OvrdCmd.1) ] OTE(Valve_XV_03.Inp_Ovrd) ] ,[P_ValveSO(Valve_XV_03) ,OTE(Valve_XV_03.Inp_NBIntlkOK) ,OTE(Valve_XV_03.Inp_IntlkOK) ] ];
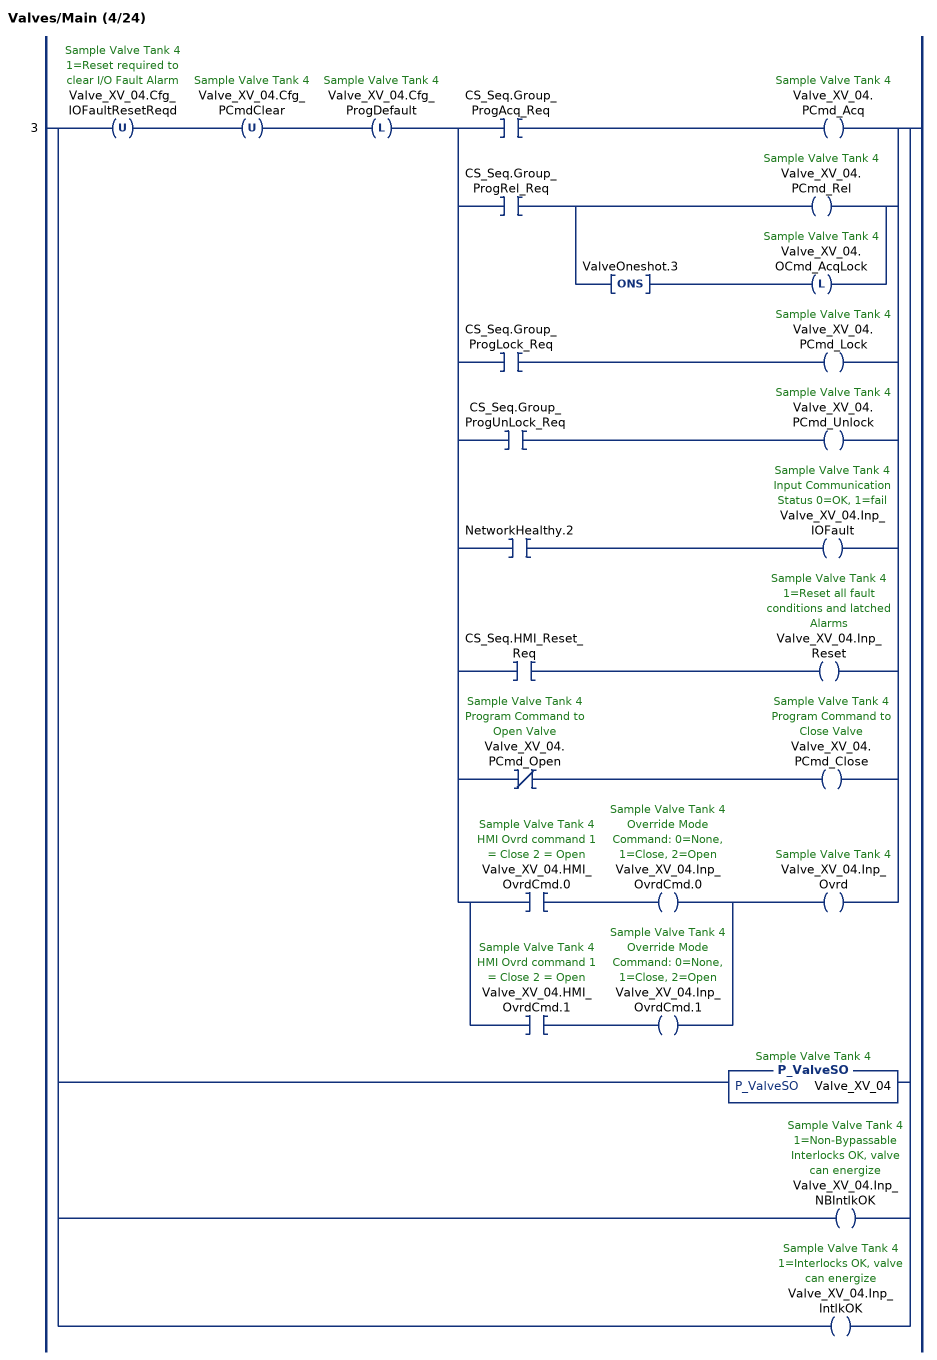
   3: [OTU(Valve_XV_04.Cfg_IOFaultResetReqd) OTU(Valve_XV_04.Cfg_PCmdClear) OTL(Valve_XV_04.Cfg_ProgDefault) [XIC(CS_Seq.Group_ProgAcq_Req) OTE(Valve_XV_04.PCmd_Acq) ,XIC(CS_Seq.Group_ProgRel_Req) [OTE(Valve_XV_04.PCmd_Rel) ,ONS(ValveOneshot.3) OTL(Valve_XV_04.OCmd_AcqLock) ] ,XIC(CS_Seq.Group_ProgLock_Req) OTE(Valve_XV_04.PCmd_Lock) ,XIC(CS_Seq.Group_ProgUnLock_Req) OTE(Valve_XV_04.PCmd_Unlock) ,XIC(NetworkHealthy.2) OTE(Valve_XV_04.Inp_IOFault) ,XIC(CS_Seq.HMI_Reset_Req) OTE(Valve_XV_04.Inp_Reset) ,XIO(Valve_XV_04.PCmd_Open) OTE(Valve_XV_04.PCmd_Close) ,[XIC(Valve_XV_04.HMI_OvrdCmd.0) OTE(Valve_XV_04.Inp_OvrdCmd.0) ,XIC(Valve_XV_04.HMI_OvrdCmd.1) OTE(Valve_XV_04.Inp_OvrdCmd.1) ] OTE(Valve_XV_04.Inp_Ovrd) ] ,[P_ValveSO(Valve_XV_04) ,OTE(Valve_XV_04.Inp_NBIntlkOK) ,OTE(Valve_XV_04.Inp_IntlkOK) ] ];
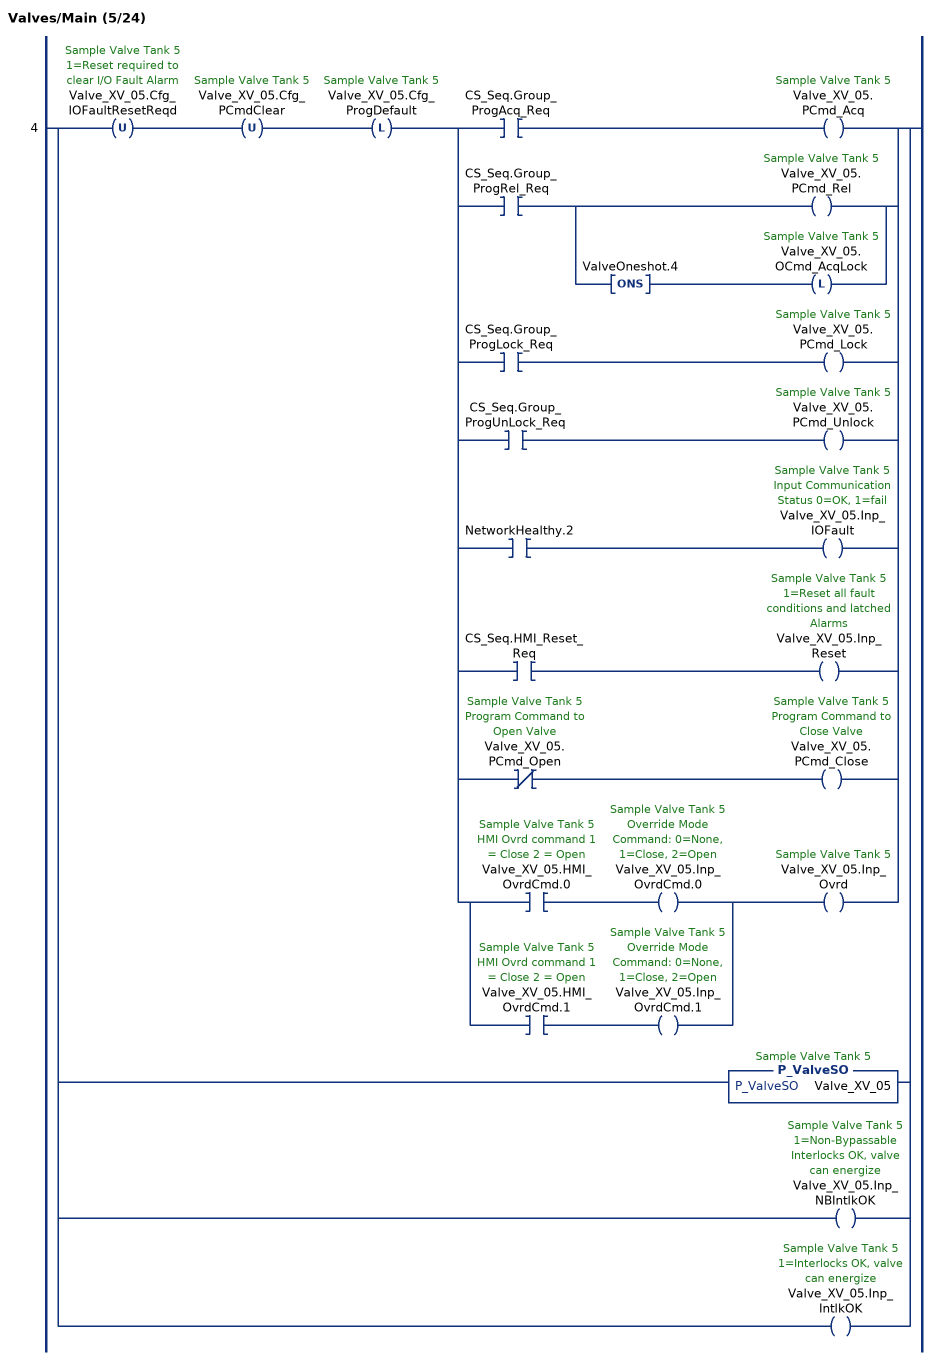
   4: [OTU(Valve_XV_05.Cfg_IOFaultResetReqd) OTU(Valve_XV_05.Cfg_PCmdClear) OTL(Valve_XV_05.Cfg_ProgDefault) [XIC(CS_Seq.Group_ProgAcq_Req) OTE(Valve_XV_05.PCmd_Acq) ,XIC(CS_Seq.Group_ProgRel_Req) [OTE(Valve_XV_05.PCmd_Rel) ,ONS(ValveOneshot.4) OTL(Valve_XV_05.OCmd_AcqLock) ] ,XIC(CS_Seq.Group_ProgLock_Req) OTE(Valve_XV_05.PCmd_Lock) ,XIC(CS_Seq.Group_ProgUnLock_Req) OTE(Valve_XV_05.PCmd_Unlock) ,XIC(NetworkHealthy.2) OTE(Valve_XV_05.Inp_IOFault) ,XIC(CS_Seq.HMI_Reset_Req) OTE(Valve_XV_05.Inp_Reset) ,XIO(Valve_XV_05.PCmd_Open) OTE(Valve_XV_05.PCmd_Close) ,[XIC(Valve_XV_05.HMI_OvrdCmd.0) OTE(Valve_XV_05.Inp_OvrdCmd.0) ,XIC(Valve_XV_05.HMI_OvrdCmd.1) OTE(Valve_XV_05.Inp_OvrdCmd.1) ] OTE(Valve_XV_05.Inp_Ovrd) ] ,[P_ValveSO(Valve_XV_05) ,OTE(Valve_XV_05.Inp_NBIntlkOK) ,OTE(Valve_XV_05.Inp_IntlkOK) ] ];
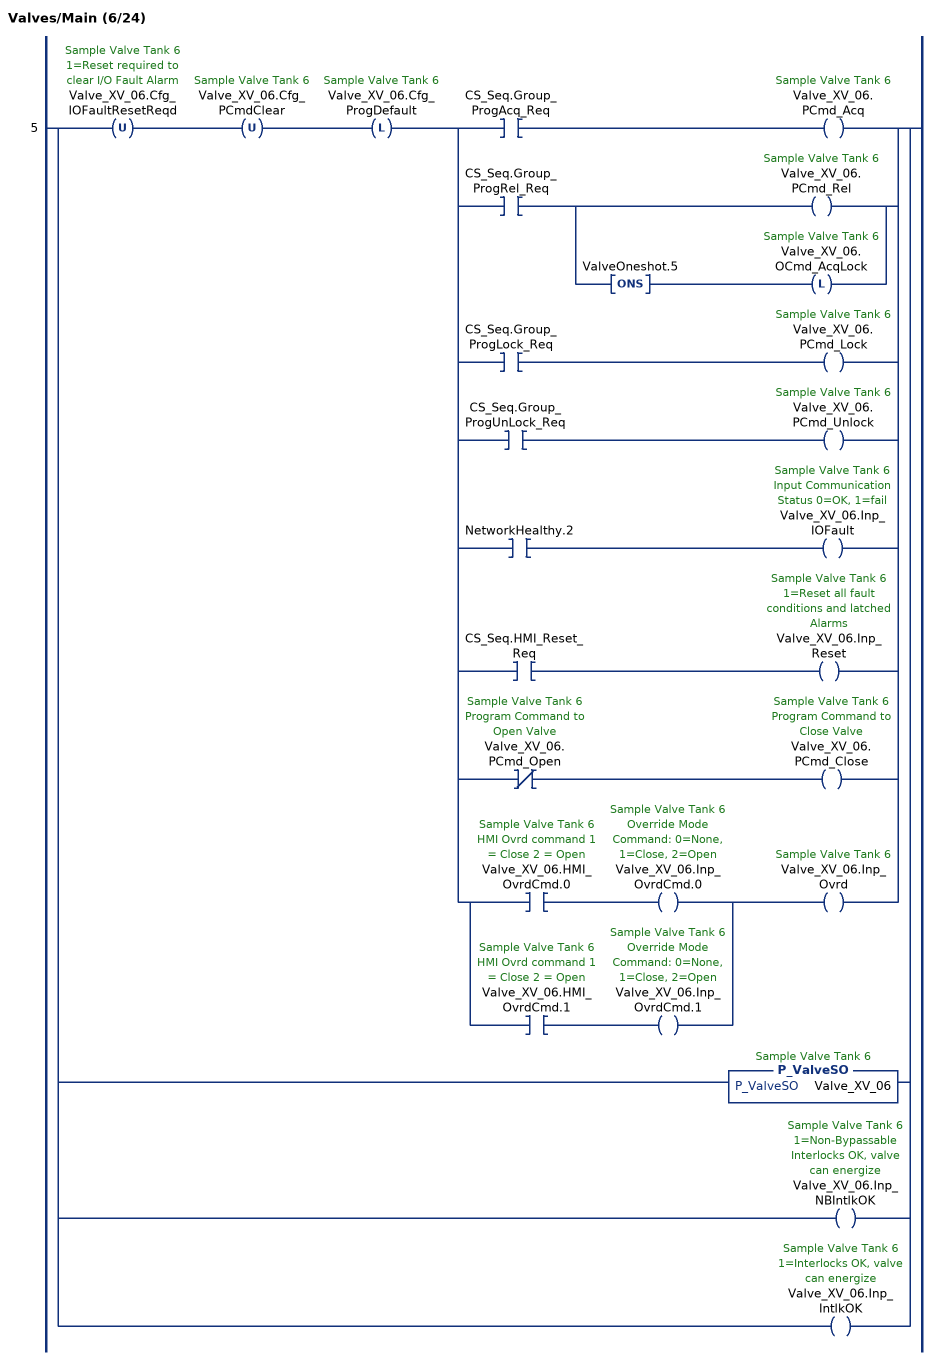
   5: [OTU(Valve_XV_06.Cfg_IOFaultResetReqd) OTU(Valve_XV_06.Cfg_PCmdClear) OTL(Valve_XV_06.Cfg_ProgDefault) [XIC(CS_Seq.Group_ProgAcq_Req) OTE(Valve_XV_06.PCmd_Acq) ,XIC(CS_Seq.Group_ProgRel_Req) [OTE(Valve_XV_06.PCmd_Rel) ,ONS(ValveOneshot.5) OTL(Valve_XV_06.OCmd_AcqLock) ] ,XIC(CS_Seq.Group_ProgLock_Req) OTE(Valve_XV_06.PCmd_Lock) ,XIC(CS_Seq.Group_ProgUnLock_Req) OTE(Valve_XV_06.PCmd_Unlock) ,XIC(NetworkHealthy.2) OTE(Valve_XV_06.Inp_IOFault) ,XIC(CS_Seq.HMI_Reset_Req) OTE(Valve_XV_06.Inp_Reset) ,XIO(Valve_XV_06.PCmd_Open) OTE(Valve_XV_06.PCmd_Close) ,[XIC(Valve_XV_06.HMI_OvrdCmd.0) OTE(Valve_XV_06.Inp_OvrdCmd.0) ,XIC(Valve_XV_06.HMI_OvrdCmd.1) OTE(Valve_XV_06.Inp_OvrdCmd.1) ] OTE(Valve_XV_06.Inp_Ovrd) ] ,[P_ValveSO(Valve_XV_06) ,OTE(Valve_XV_06.Inp_NBIntlkOK) ,OTE(Valve_XV_06.Inp_IntlkOK) ] ];
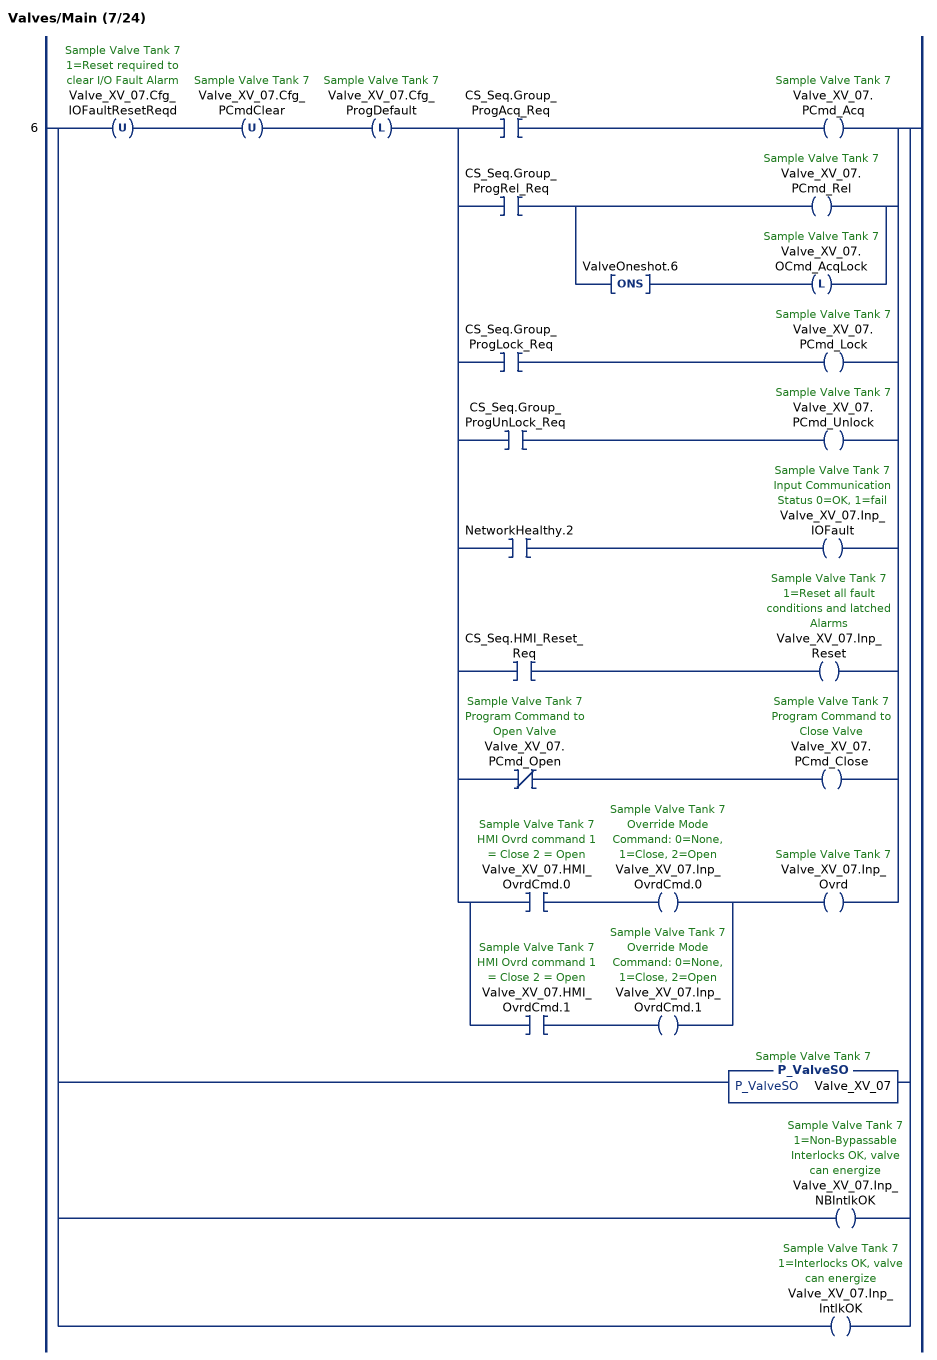
   6: [OTU(Valve_XV_07.Cfg_IOFaultResetReqd) OTU(Valve_XV_07.Cfg_PCmdClear) OTL(Valve_XV_07.Cfg_ProgDefault) [XIC(CS_Seq.Group_ProgAcq_Req) OTE(Valve_XV_07.PCmd_Acq) ,XIC(CS_Seq.Group_ProgRel_Req) [OTE(Valve_XV_07.PCmd_Rel) ,ONS(ValveOneshot.6) OTL(Valve_XV_07.OCmd_AcqLock) ] ,XIC(CS_Seq.Group_ProgLock_Req) OTE(Valve_XV_07.PCmd_Lock) ,XIC(CS_Seq.Group_ProgUnLock_Req) OTE(Valve_XV_07.PCmd_Unlock) ,XIC(NetworkHealthy.2) OTE(Valve_XV_07.Inp_IOFault) ,XIC(CS_Seq.HMI_Reset_Req) OTE(Valve_XV_07.Inp_Reset) ,XIO(Valve_XV_07.PCmd_Open) OTE(Valve_XV_07.PCmd_Close) ,[XIC(Valve_XV_07.HMI_OvrdCmd.0) OTE(Valve_XV_07.Inp_OvrdCmd.0) ,XIC(Valve_XV_07.HMI_OvrdCmd.1) OTE(Valve_XV_07.Inp_OvrdCmd.1) ] OTE(Valve_XV_07.Inp_Ovrd) ] ,[P_ValveSO(Valve_XV_07) ,OTE(Valve_XV_07.Inp_NBIntlkOK) ,OTE(Valve_XV_07.Inp_IntlkOK) ] ];
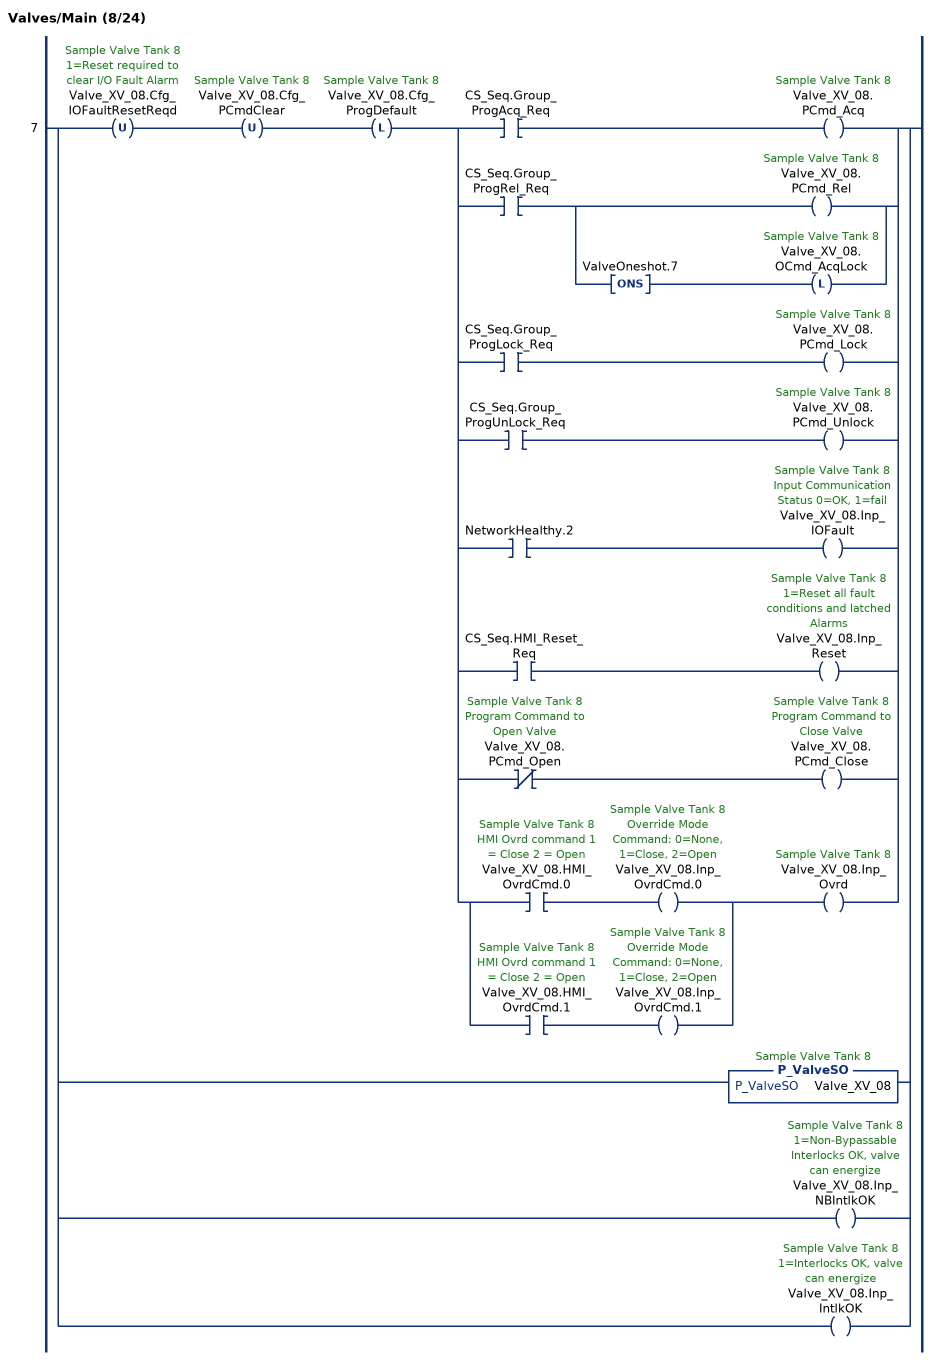
   7: [OTU(Valve_XV_08.Cfg_IOFaultResetReqd) OTU(Valve_XV_08.Cfg_PCmdClear) OTL(Valve_XV_08.Cfg_ProgDefault) [XIC(CS_Seq.Group_ProgAcq_Req) OTE(Valve_XV_08.PCmd_Acq) ,XIC(CS_Seq.Group_ProgRel_Req) [OTE(Valve_XV_08.PCmd_Rel) ,ONS(ValveOneshot.7) OTL(Valve_XV_08.OCmd_AcqLock) ] ,XIC(CS_Seq.Group_ProgLock_Req) OTE(Valve_XV_08.PCmd_Lock) ,XIC(CS_Seq.Group_ProgUnLock_Req) OTE(Valve_XV_08.PCmd_Unlock) ,XIC(NetworkHealthy.2) OTE(Valve_XV_08.Inp_IOFault) ,XIC(CS_Seq.HMI_Reset_Req) OTE(Valve_XV_08.Inp_Reset) ,XIO(Valve_XV_08.PCmd_Open) OTE(Valve_XV_08.PCmd_Close) ,[XIC(Valve_XV_08.HMI_OvrdCmd.0) OTE(Valve_XV_08.Inp_OvrdCmd.0) ,XIC(Valve_XV_08.HMI_OvrdCmd.1) OTE(Valve_XV_08.Inp_OvrdCmd.1) ] OTE(Valve_XV_08.Inp_Ovrd) ] ,[P_ValveSO(Valve_XV_08) ,OTE(Valve_XV_08.Inp_NBIntlkOK) ,OTE(Valve_XV_08.Inp_IntlkOK) ] ];
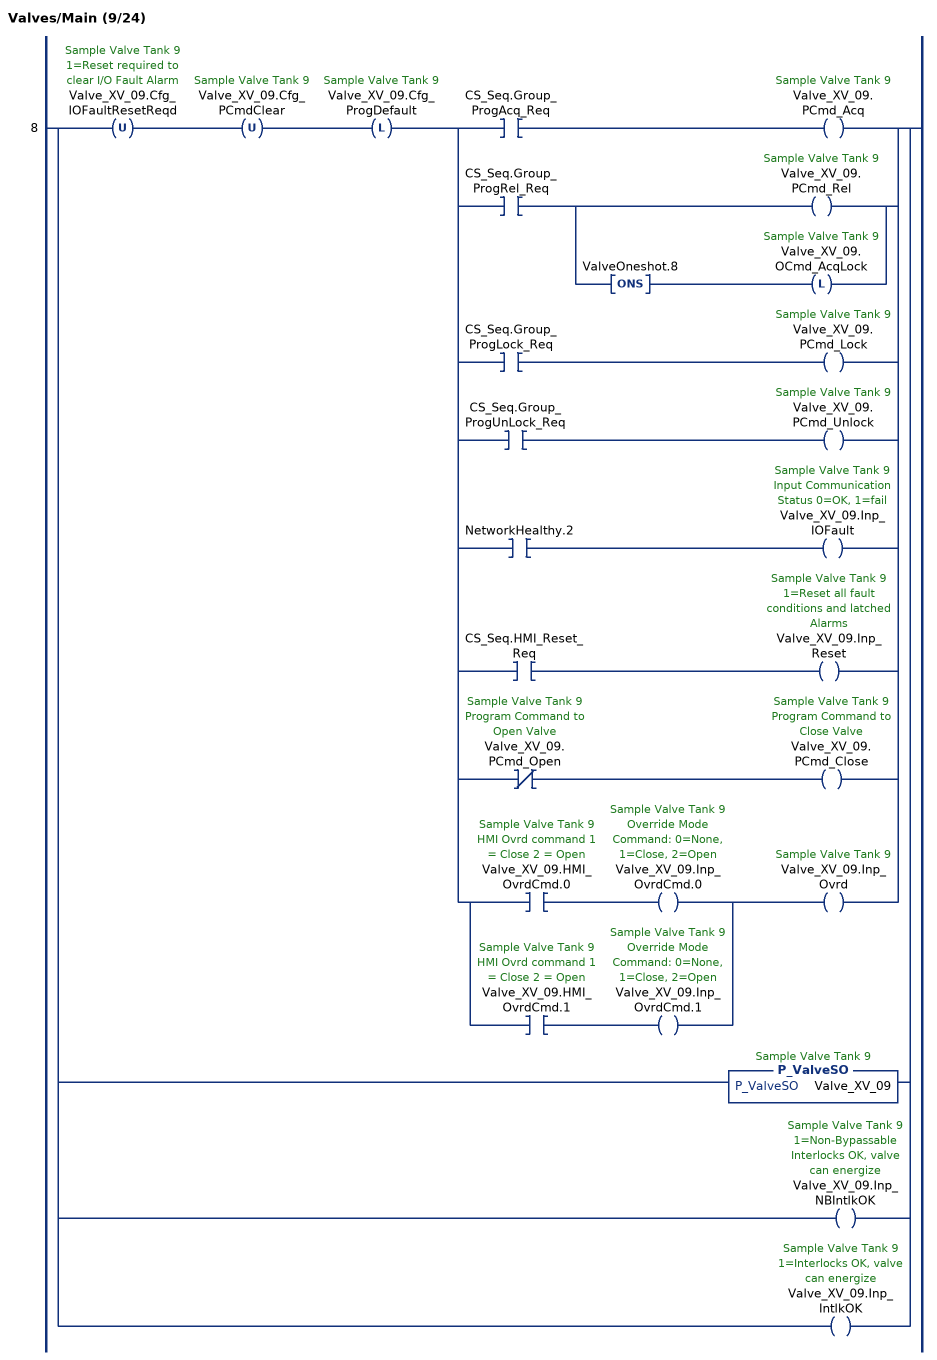
   8: [OTU(Valve_XV_09.Cfg_IOFaultResetReqd) OTU(Valve_XV_09.Cfg_PCmdClear) OTL(Valve_XV_09.Cfg_ProgDefault) [XIC(CS_Seq.Group_ProgAcq_Req) OTE(Valve_XV_09.PCmd_Acq) ,XIC(CS_Seq.Group_ProgRel_Req) [OTE(Valve_XV_09.PCmd_Rel) ,ONS(ValveOneshot.8) OTL(Valve_XV_09.OCmd_AcqLock) ] ,XIC(CS_Seq.Group_ProgLock_Req) OTE(Valve_XV_09.PCmd_Lock) ,XIC(CS_Seq.Group_ProgUnLock_Req) OTE(Valve_XV_09.PCmd_Unlock) ,XIC(NetworkHealthy.2) OTE(Valve_XV_09.Inp_IOFault) ,XIC(CS_Seq.HMI_Reset_Req) OTE(Valve_XV_09.Inp_Reset) ,XIO(Valve_XV_09.PCmd_Open) OTE(Valve_XV_09.PCmd_Close) ,[XIC(Valve_XV_09.HMI_OvrdCmd.0) OTE(Valve_XV_09.Inp_OvrdCmd.0) ,XIC(Valve_XV_09.HMI_OvrdCmd.1) OTE(Valve_XV_09.Inp_OvrdCmd.1) ] OTE(Valve_XV_09.Inp_Ovrd) ] ,[P_ValveSO(Valve_XV_09) ,OTE(Valve_XV_09.Inp_NBIntlkOK) ,OTE(Valve_XV_09.Inp_IntlkOK) ] ];
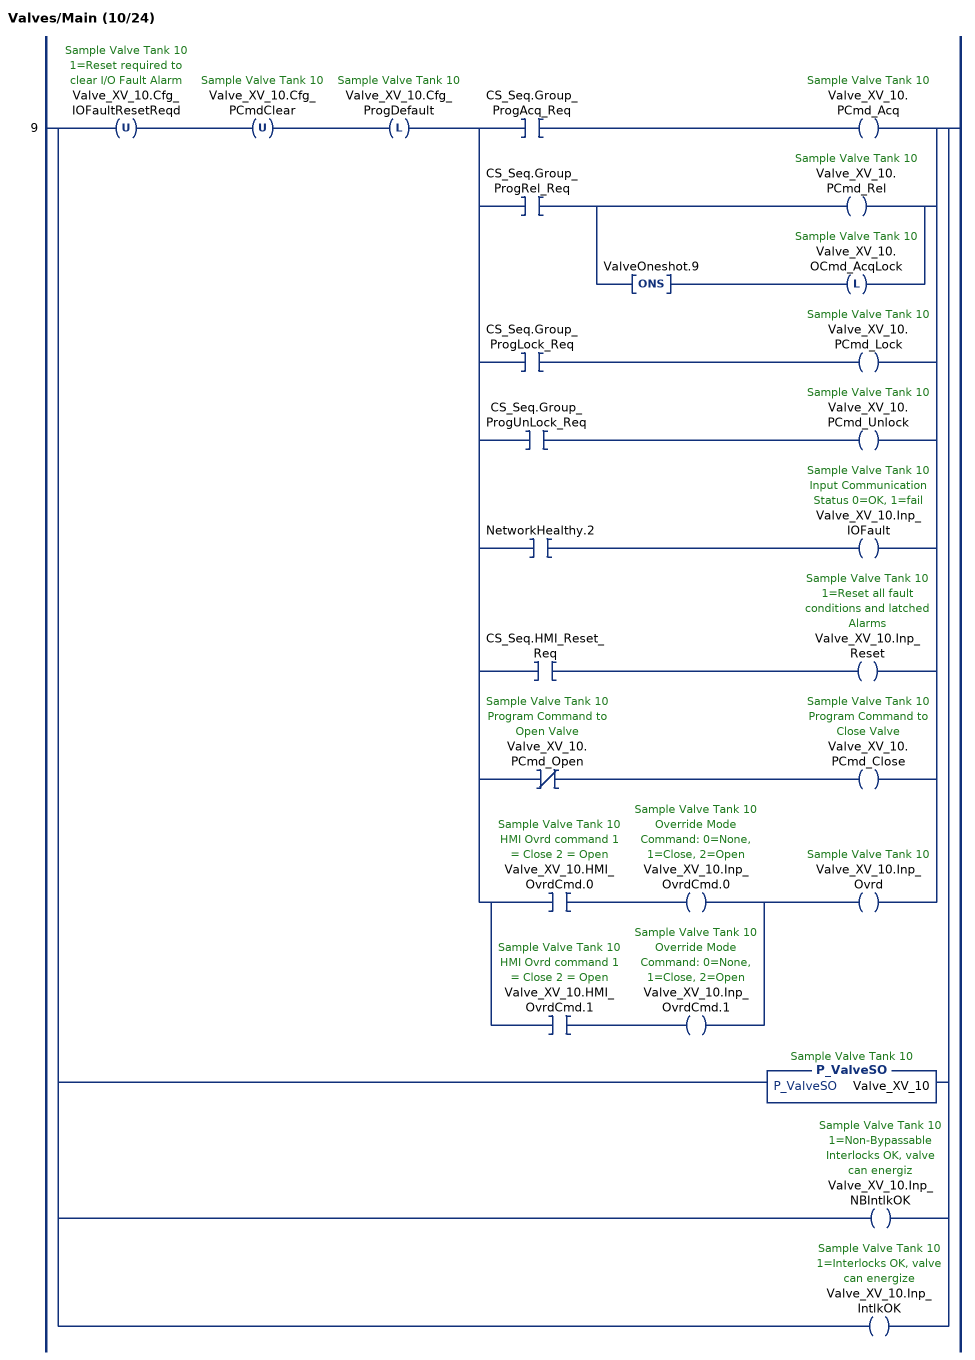
   9: [OTU(Valve_XV_10.Cfg_IOFaultResetReqd) OTU(Valve_XV_10.Cfg_PCmdClear) OTL(Valve_XV_10.Cfg_ProgDefault) [XIC(CS_Seq.Group_ProgAcq_Req) OTE(Valve_XV_10.PCmd_Acq) ,XIC(CS_Seq.Group_ProgRel_Req) [OTE(Valve_XV_10.PCmd_Rel) ,ONS(ValveOneshot.9) OTL(Valve_XV_10.OCmd_AcqLock) ] ,XIC(CS_Seq.Group_ProgLock_Req) OTE(Valve_XV_10.PCmd_Lock) ,XIC(CS_Seq.Group_ProgUnLock_Req) OTE(Valve_XV_10.PCmd_Unlock) ,XIC(NetworkHealthy.2) OTE(Valve_XV_10.Inp_IOFault) ,XIC(CS_Seq.HMI_Reset_Req) OTE(Valve_XV_10.Inp_Reset) ,XIO(Valve_XV_10.PCmd_Open) OTE(Valve_XV_10.PCmd_Close) ,[XIC(Valve_XV_10.HMI_OvrdCmd.0) OTE(Valve_XV_10.Inp_OvrdCmd.0) ,XIC(Valve_XV_10.HMI_OvrdCmd.1) OTE(Valve_XV_10.Inp_OvrdCmd.1) ] OTE(Valve_XV_10.Inp_Ovrd) ] ,[P_ValveSO(Valve_XV_10) ,OTE(Valve_XV_10.Inp_NBIntlkOK) ,OTE(Valve_XV_10.Inp_IntlkOK) ] ];
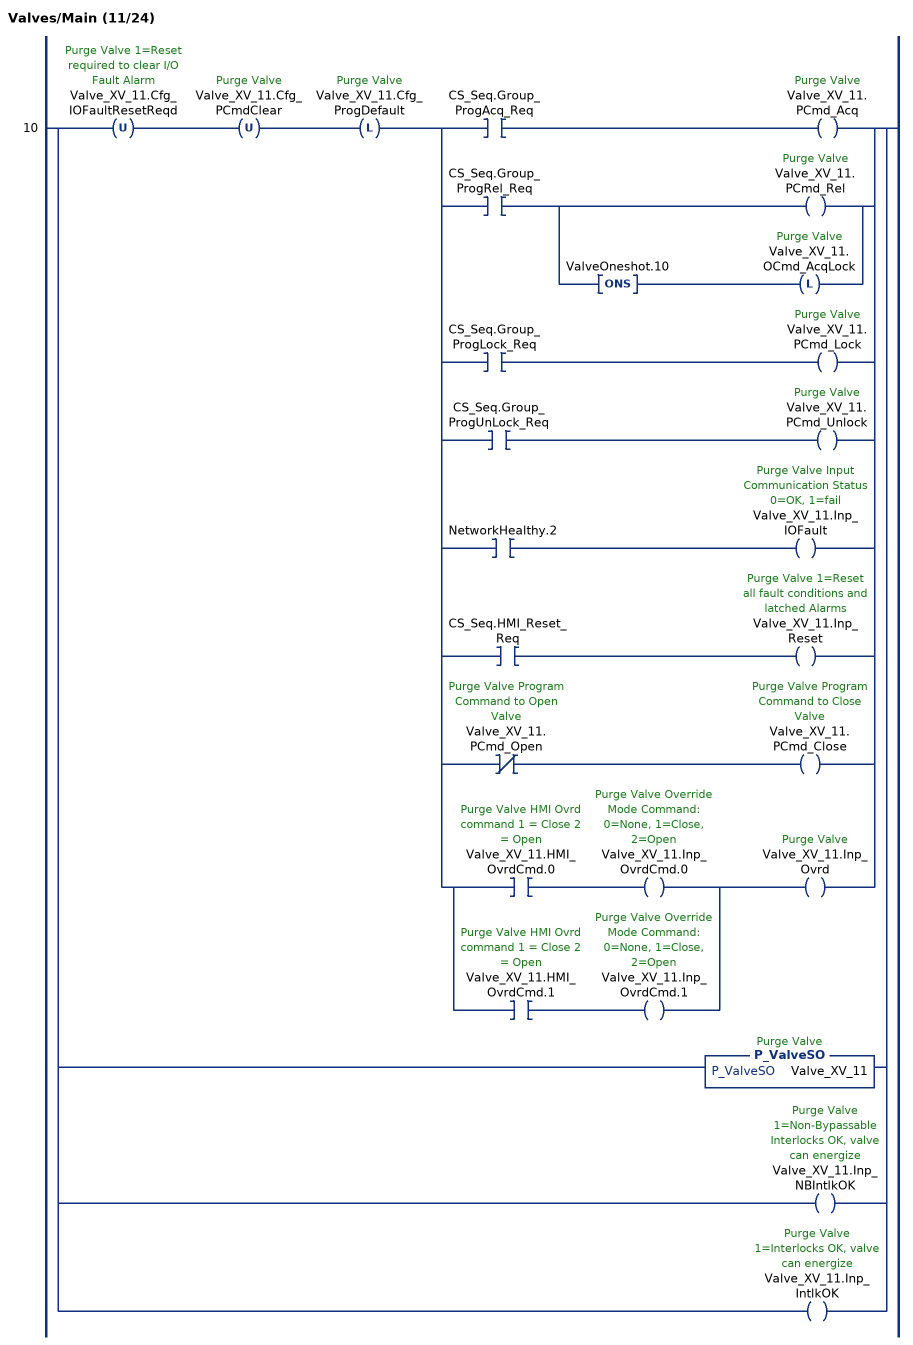
   10: [OTU(Valve_XV_11.Cfg_IOFaultResetReqd) OTU(Valve_XV_11.Cfg_PCmdClear) OTL(Valve_XV_11.Cfg_ProgDefault) [XIC(CS_Seq.Group_ProgAcq_Req) OTE(Valve_XV_11.PCmd_Acq) ,XIC(CS_Seq.Group_ProgRel_Req) [OTE(Valve_XV_11.PCmd_Rel) ,ONS(ValveOneshot.10) OTL(Valve_XV_11.OCmd_AcqLock) ] ,XIC(CS_Seq.Group_ProgLock_Req) OTE(Valve_XV_11.PCmd_Lock) ,XIC(CS_Seq.Group_ProgUnLock_Req) OTE(Valve_XV_11.PCmd_Unlock) ,XIC(NetworkHealthy.2) OTE(Valve_XV_11.Inp_IOFault) ,XIC(CS_Seq.HMI_Reset_Req) OTE(Valve_XV_11.Inp_Reset) ,XIO(Valve_XV_11.PCmd_Open) OTE(Valve_XV_11.PCmd_Close) ,[XIC(Valve_XV_11.HMI_OvrdCmd.0) OTE(Valve_XV_11.Inp_OvrdCmd.0) ,XIC(Valve_XV_11.HMI_OvrdCmd.1) OTE(Valve_XV_11.Inp_OvrdCmd.1) ] OTE(Valve_XV_11.Inp_Ovrd) ] ,[P_ValveSO(Valve_XV_11) ,OTE(Valve_XV_11.Inp_NBIntlkOK) ,OTE(Valve_XV_11.Inp_IntlkOK) ] ];
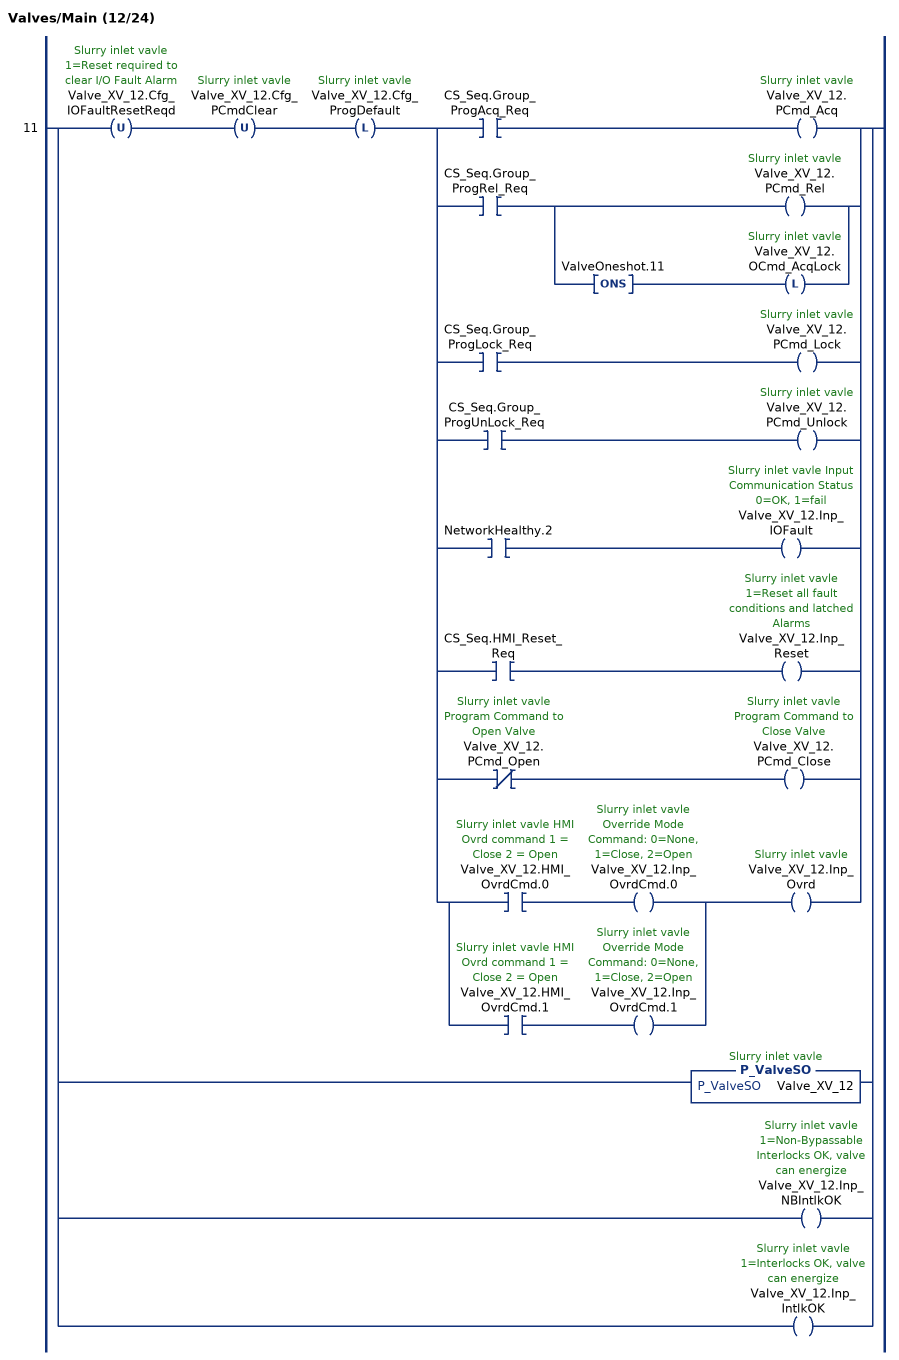
   11: [OTU(Valve_XV_12.Cfg_IOFaultResetReqd) OTU(Valve_XV_12.Cfg_PCmdClear) OTL(Valve_XV_12.Cfg_ProgDefault) [XIC(CS_Seq.Group_ProgAcq_Req) OTE(Valve_XV_12.PCmd_Acq) ,XIC(CS_Seq.Group_ProgRel_Req) [OTE(Valve_XV_12.PCmd_Rel) ,ONS(ValveOneshot.11) OTL(Valve_XV_12.OCmd_AcqLock) ] ,XIC(CS_Seq.Group_ProgLock_Req) OTE(Valve_XV_12.PCmd_Lock) ,XIC(CS_Seq.Group_ProgUnLock_Req) OTE(Valve_XV_12.PCmd_Unlock) ,XIC(NetworkHealthy.2) OTE(Valve_XV_12.Inp_IOFault) ,XIC(CS_Seq.HMI_Reset_Req) OTE(Valve_XV_12.Inp_Reset) ,XIO(Valve_XV_12.PCmd_Open) OTE(Valve_XV_12.PCmd_Close) ,[XIC(Valve_XV_12.HMI_OvrdCmd.0) OTE(Valve_XV_12.Inp_OvrdCmd.0) ,XIC(Valve_XV_12.HMI_OvrdCmd.1) OTE(Valve_XV_12.Inp_OvrdCmd.1) ] OTE(Valve_XV_12.Inp_Ovrd) ] ,[P_ValveSO(Valve_XV_12) ,OTE(Valve_XV_12.Inp_NBIntlkOK) ,OTE(Valve_XV_12.Inp_IntlkOK) ] ];
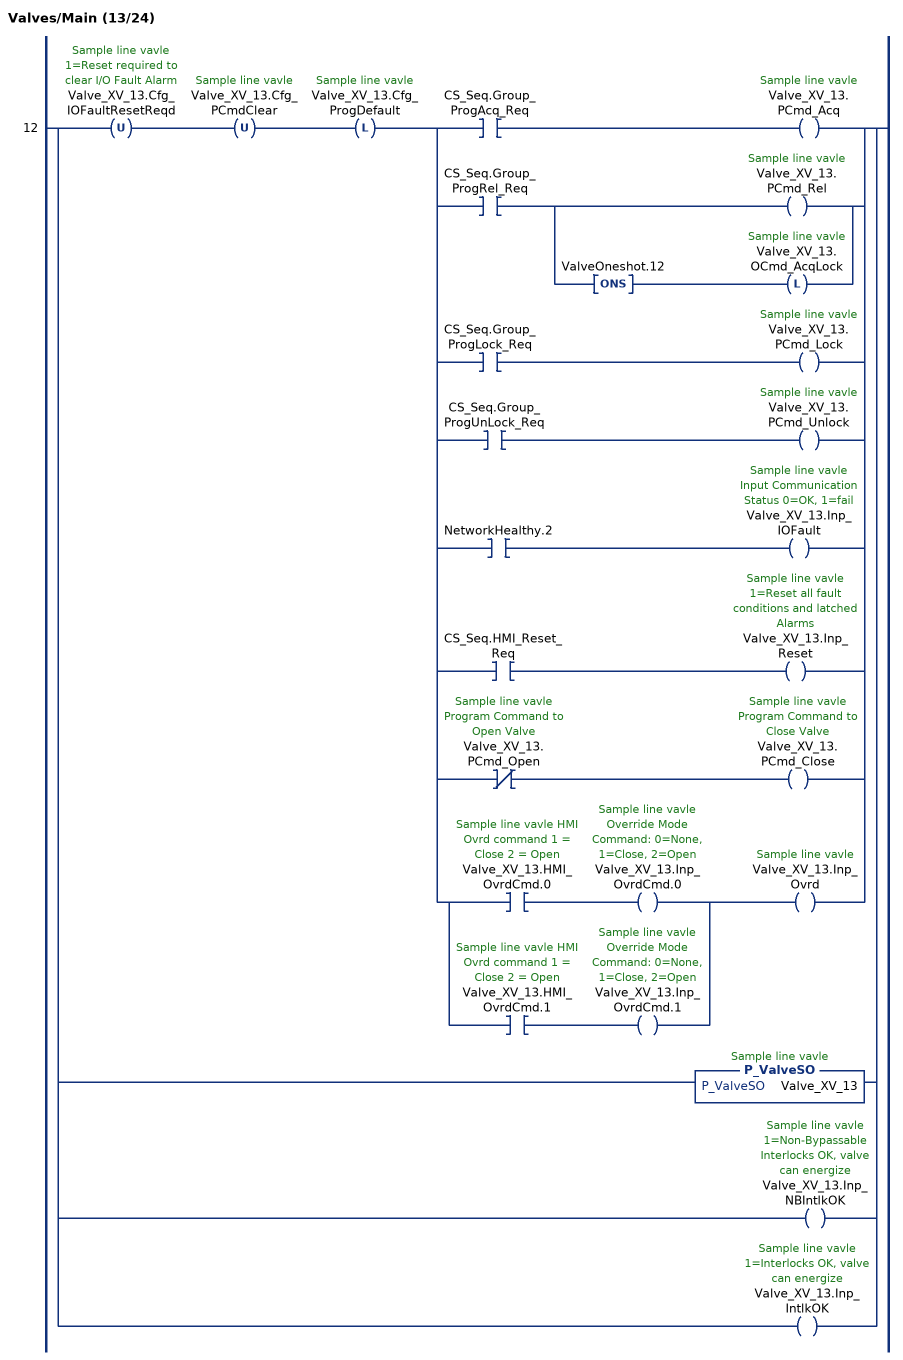
   12: [OTU(Valve_XV_13.Cfg_IOFaultResetReqd) OTU(Valve_XV_13.Cfg_PCmdClear) OTL(Valve_XV_13.Cfg_ProgDefault) [XIC(CS_Seq.Group_ProgAcq_Req) OTE(Valve_XV_13.PCmd_Acq) ,XIC(CS_Seq.Group_ProgRel_Req) [OTE(Valve_XV_13.PCmd_Rel) ,ONS(ValveOneshot.12) OTL(Valve_XV_13.OCmd_AcqLock) ] ,XIC(CS_Seq.Group_ProgLock_Req) OTE(Valve_XV_13.PCmd_Lock) ,XIC(CS_Seq.Group_ProgUnLock_Req) OTE(Valve_XV_13.PCmd_Unlock) ,XIC(NetworkHealthy.2) OTE(Valve_XV_13.Inp_IOFault) ,XIC(CS_Seq.HMI_Reset_Req) OTE(Valve_XV_13.Inp_Reset) ,XIO(Valve_XV_13.PCmd_Open) OTE(Valve_XV_13.PCmd_Close) ,[XIC(Valve_XV_13.HMI_OvrdCmd.0) OTE(Valve_XV_13.Inp_OvrdCmd.0) ,XIC(Valve_XV_13.HMI_OvrdCmd.1) OTE(Valve_XV_13.Inp_OvrdCmd.1) ] OTE(Valve_XV_13.Inp_Ovrd) ] ,[P_ValveSO(Valve_XV_13) ,OTE(Valve_XV_13.Inp_NBIntlkOK) ,OTE(Valve_XV_13.Inp_IntlkOK) ] ];
